Universal Robots PolyScope program: DAS428_958_02_MAR_21_DAS_lado_izquierdo_jig2.urp

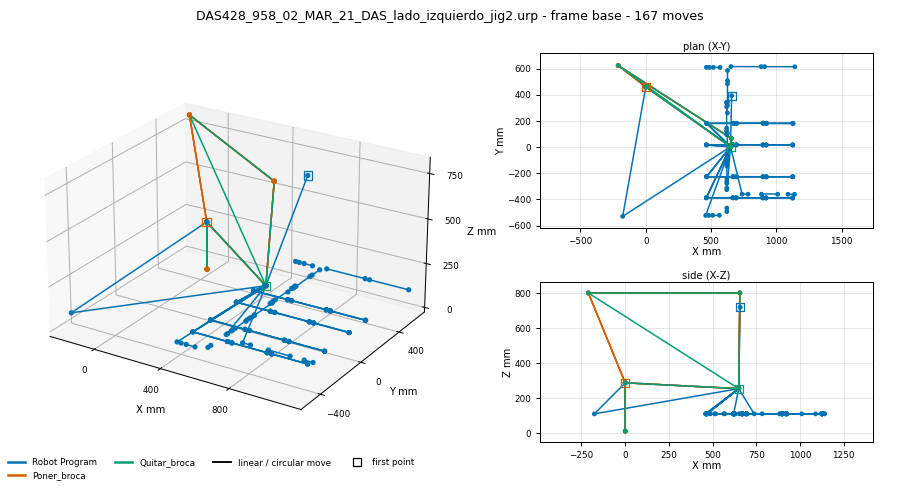
[picture p0: tool path of DAS428_958_02_MAR_21_DAS_lado_izquierdo_jig2.urp in frame base, 167 of 340 moves have a stored position in this frame; points joined in program order, loops and branches not executed]
Program DAS428_958_02_MAR_21_DAS_lado_izquierdo_jig2 (installation=instalacion_derecha_10_MAR_21 directory=/programs/jig2/Izquierda createdIn=5.6.0.90886 lastSavedIn=5.6.0.90886 robotSerialNumber=20195001785)
Calibrated DH parameters: a=[0.000107, -0.568984, -0.552934, -0.00001, -0.000063, 0]; d=[0.180718, -257.998067, 200.685024, 57.48776, 0.119923, 0.115353]; alpha=[1.571119, 0.000876, -0.002498, 1.571178, -1.570523, 0]; deltaTheta=[0, -0.378191, 0.631587, -0.253396, 0, 0]
Robot Program (runOnlyOnce=false)
  Folder Variables
    bajada_broca := p[0,0,-0.008,0,0,0]
    barrenos_menos1 := 0
    barreno_actual := 0
    posicion := p[0,0,300,0,0,0]
    cambiar_broca := False
    barrenos_hechos := 0
    eje7 := 0
    Wait Sleep waitTime=0.5
  Folder Home
    Wait Sleep waitTime=0.3
    MoveL speed 250 mm/s, acceleration 1200 mm/s^2 (useActiveTCP=true) feature=Base
      Waypoint Traslacion: TCP in base x=657.999 y=394.119 z=719.669 mm, rx=0.7459 ry=2.9065 rz=0.0955 rad; joints [-173.083, -83.201, 56.688, 18.113, -333.312, 0.041] deg; TCP offset x=0.411 y=-218.298 z=37.994 mm, rx=1.558 ry=-0.1255 rz=0.1212 rad
      Waypoint Home2: TCP in base x=649.602 y=3.2 z=254.15 mm, rx=-2.4485 ry=-1.9662 rz=-0.0111 rad; joints [-199.372, -96.579, 116.673, -19.801, -286.041, 0.348] deg; TCP offset x=0.411 y=-218.298 z=37.994 mm, rx=1.558 ry=-0.1255 rz=0.1212 rad
      Waypoint Home3: TCP in base x=649.602 y=3.2 z=254.15 mm, rx=-2.4485 ry=-1.9662 rz=-0.0111 rad; joints [-199.372, -96.579, 116.673, -19.801, -286.041, 0.348] deg; TCP offset x=0.411 y=-218.298 z=37.994 mm, rx=1.558 ry=-0.1255 rz=0.1212 rad
      Waypoint Home4: TCP in base x=649.602 y=3.2 z=254.15 mm, rx=-2.4485 ry=-1.9662 rz=-0.0111 rad; joints [-199.372, -96.579, 116.673, -19.801, -286.041, 0.348] deg
      Waypoint PosicionApagado: TCP in base x=-175.961 y=-529.389 z=109.95 mm, rx=0.175 ry=2.1133 rz=-2.1574 rad; joints [-90.111, -89.982, -160.832, -17.508, -269.675, 0.001] deg; TCP offset x=0.411 y=-218.298 z=37.994 mm, rx=1.558 ry=-0.1255 rz=0.1212 rad
      Waypoint Precambio_broca: TCP in base x=0.83 y=461.518 z=287.521 mm, rx=-0.2218 ry=-3.132 rz=0.0004 rad; joints [-125.124, -120.118, 128.54, -7.699, -306.118, -0.232] deg
    SafeHome (positionOptionType=SPEED_AND_ACCELERATION speed=1.047198 acceleration=1.396263 nextMotionTime=2)
    SuppressedNode
      MoveL speed 250 mm/s, acceleration 1200 mm/s^2 (useActiveTCP=true) feature=Base
        Waypoint home_trans: TCP in base x=-171.077 y=546.65 z=109.574 mm, rx=0.1544 ry=3.1247 rz=-0.2011 rad; joints [-91.802, -93.053, 127.954, -27.005, -275.278, -0.192] deg
    Wait Sleep waitTime=0.3
    iniciando_prog := True
    Call Poner_broca
  Folder Posicion2
    Folder Inicio
      eje7 := 2
      MoveL speed 250 mm/s, acceleration 1200 mm/s^2 (useActiveTCP=true) feature=Base
        Waypoint Home2: TCP in base x=649.602 y=3.2 z=254.15 mm, rx=-2.4485 ry=-1.9662 rz=-0.0111 rad; joints [-199.372, -96.579, 116.673, -19.801, -286.041, 0.348] deg; TCP offset x=0.411 y=-218.298 z=37.994 mm, rx=1.558 ry=-0.1255 rz=0.1212 rad
    Folder SeatTracks
      Folder Broca_1
        Folder Linea1
          Folder Marcar_puntos
            MoveL speed 100 mm/s, acceleration 500 mm/s^2 (useActiveTCP=true) feature=Base
              Waypoint Home2: TCP in base x=649.602 y=3.2 z=254.15 mm, rx=-2.4485 ry=-1.9662 rz=-0.0111 rad; joints [-199.372, -96.579, 116.673, -19.801, -286.041, 0.348] deg
              Waypoint Linea1_A: TCP in base x=465.78 y=-226.285 z=110.11 mm, rx=3.1292 ry=0.274 rz=-0.0085 rad; joints [-215.56, -96.678, 133.119, -35.816, -234.732, 0.192] deg; TCP offset x=0.411 y=-218.298 z=37.994 mm, rx=1.558 ry=-0.1255 rz=0.1212 rad
              Waypoint Linea1_B: TCP in base x=669.2 y=-226.066 z=110.222 mm, rx=3.1292 ry=0.2741 rz=-0.0085 rad; joints [-203.814, -77.304, 112.388, -34.338, -222.994, 0.395] deg; TCP offset x=0.411 y=-218.298 z=37.994 mm, rx=1.558 ry=-0.1255 rz=0.1212 rad
              Waypoint Linea1_C: TCP in base x=694.6 y=-226.083 z=110.775 mm, rx=3.1292 ry=0.274 rz=-0.0086 rad; joints [-202.875, -75.175, 109.532, -33.596, -222.053, 0.413] deg
              Waypoint Linea1_D: TCP in base x=897.8 y=-226.331 z=110.549 mm, rx=3.1292 ry=0.2741 rz=-0.0085 rad; joints [-197.398, -58.161, 84.21, -25.204, -216.564, 0.534] deg
              Waypoint Linea1_E: TCP in base x=923.2 y=-226.496 z=110.279 mm, rx=3.1292 ry=0.2741 rz=-0.0086 rad; joints [-196.902, -55.941, 80.587, -23.787, -216.064, 0.545] deg
              Waypoint Linea1_F: TCP in base x=1125.593 y=-226.031 z=110.602 mm, rx=3.1292 ry=0.2741 rz=-0.0087 rad; joints [-193.7, -34.945, 43.134, -7.265, -212.819, 0.625] deg; TCP offset x=0.411 y=-218.298 z=37.994 mm, rx=1.558 ry=-0.1255 rz=0.1212 rad
          Folder AB
            'desbaste_inicial'
            bajada_broca := p[0,0,-0.008,0,0,0]
            barrenos_menos1 := 8
            barreno_actual := 0
            Loop While (checkContinuously=false) expression=barreno_actual≤barrenos_menos1
              Folder Perforacion
                MoveL speed 100 mm/s, acceleration 500 mm/s^2 (useActiveTCP=true) feature=Base
                  internos := interpolate_pose(Linea1_A, Linea1_B, barreno_actual/barrenos_menos1)
                  Waypoint Waypoint (Variable): variable=internos
                  'desbaste_inicial'
                  bajada_broca := p[0,0,-0.008,0,0,0]
                  bajada := p[0,0,0.008,0,0,0]
                  MoveDirectionNode (selectedDirection=ZMinus toolParams=0.015, 0.015)
                    Until DISTANCE (allowActions=false deceleration=3 distanceNodeType=STOP) Distance=0.076; motionParameters(blendRadius=0)
                  Popup Message (haltProgram=false message=punto contacto alanzdo inputType=Text)
                  MoveDirectionNode (selectedDirection=ZPlus toolParams=0.015, 0.015)
                    Until DISTANCE (allowActions=false deceleration=3 distanceNodeType=STOP) Distance=0.002; motionParameters(blendRadius=0)
                  Wait Sleep waitTime=0.3
                  Set DigitalOutput pin=config_out[1]; digitalValue=1
                  Wait Sleep waitTime=0.3
                  Loop Counting (count=3) loopVariable(name=Loop_39)
                    bajar := pose_add(get_actual_tcp_pose(), bajada_broca)
                    Waypoint Waypoint (Variable): motionParameters(jointSpeed=1.047198 jointAcceleration=1.396263 cartesianSpeed=0.001 cartesianAcceleration=0.005); variable=bajar
                    subir := pose_sub(get_actual_tcp_pose(), bajada_broca)
                    Waypoint Waypoint (Variable): motionParameters(jointSpeed=1.047198 jointAcceleration=1.396263 cartesianSpeed=0.005 cartesianAcceleration=0.01); variable=subir
                    bajada_broca := pose_sub(bajada_broca, bajada)
                  MoveDirectionNode (selectedDirection=ZPlus toolParams=0.03, 0.035)
                    Until DISTANCE (allowActions=false deceleration=3 distanceNodeType=STOP) Distance=0.06; motionParameters(blendRadius=0)
                  Set DigitalOutput pin=config_out[1]; digitalValue=0
                  barreno_actual := barreno_actual+1
                  SuppressedNode
                    Call Quitar_broca
                  SuppressedNode
                    Call Poner_broca
          Folder CD
            'desbaste_inicial'
            bajada_broca := p[0,0,-0.008,0,0,0]
            barrenos_menos1 := 8
            barreno_actual := 0
            Loop While (checkContinuously=false) expression=barreno_actual≤barrenos_menos1
              Folder Perforacion
                MoveL speed 100 mm/s, acceleration 500 mm/s^2 (useActiveTCP=true) feature=Base
                  internos := interpolate_pose(Linea1_C, Linea1_D, barreno_actual/barrenos_menos1)
                  Waypoint Waypoint (Variable): variable=internos
                  'desbaste_inicial'
                  bajada_broca := p[0,0,-0.008,0,0,0]
                  bajada := p[0,0,0.008,0,0,0]
                  MoveDirectionNode (selectedDirection=ZMinus toolParams=0.015, 0.015)
                    Until DISTANCE (allowActions=false deceleration=3 distanceNodeType=STOP) Distance=0.076; motionParameters(blendRadius=0)
                  Popup Message (haltProgram=false message=punto contacto alanzdo inputType=Text)
                  MoveDirectionNode (selectedDirection=ZPlus toolParams=0.003, 0.005)
                    Until DISTANCE (allowActions=false deceleration=3 distanceNodeType=STOP) Distance=0.002; motionParameters(blendRadius=0)
                  Wait Sleep waitTime=0.3
                  Set DigitalOutput pin=config_out[1]; digitalValue=1
                  Wait Sleep waitTime=0.3
                  Loop Counting (count=3) loopVariable(name=Loop_56)
                    bajar := pose_add(get_actual_tcp_pose(), bajada_broca)
                    Waypoint Waypoint (Variable): motionParameters(jointSpeed=1.047198 jointAcceleration=1.396263 cartesianSpeed=0.001 cartesianAcceleration=0.005); variable=bajar
                    subir := pose_sub(get_actual_tcp_pose(), bajada_broca)
                    Waypoint Waypoint (Variable): motionParameters(jointSpeed=1.047198 jointAcceleration=1.396263 cartesianSpeed=0.005 cartesianAcceleration=0.01); variable=subir
                    bajada_broca := pose_sub(bajada_broca, bajada)
                  MoveDirectionNode (selectedDirection=ZPlus toolParams=0.03, 0.035)
                    Until DISTANCE (allowActions=false deceleration=3 distanceNodeType=STOP) Distance=0.06; motionParameters(blendRadius=0)
                  Set DigitalOutput pin=config_out[1]; digitalValue=0
                  barreno_actual := barreno_actual+1
                  SuppressedNode
                    Call Quitar_broca
                  SuppressedNode
                    Call Poner_broca
          Folder EF
            'desbaste_inicial'
            bajada_broca := p[0,0,-0.008,0,0,0]
            barrenos_menos1 := 8
            barreno_actual := 0
            Loop While (checkContinuously=false) expression=barreno_actual≤barrenos_menos1
              Folder Perforacion
                MoveL speed 100 mm/s, acceleration 500 mm/s^2 (useActiveTCP=true) feature=Base
                  internos := interpolate_pose(Linea1_E, Linea1_F, barreno_actual/barrenos_menos1)
                  Waypoint Waypoint (Variable): variable=internos
                  'desbaste_inicial'
                  bajada_broca := p[0,0,-0.008,0,0,0]
                  bajada := p[0,0,0.008,0,0,0]
                  MoveDirectionNode (selectedDirection=ZMinus toolParams=0.015, 0.015)
                    Until DISTANCE (allowActions=false deceleration=3 distanceNodeType=STOP) Distance=0.076; motionParameters(blendRadius=0)
                  Popup Message (haltProgram=false message=punto contacto alanzdo inputType=Text)
                  MoveDirectionNode (selectedDirection=ZPlus toolParams=0.003, 0.005)
                    Until DISTANCE (allowActions=false deceleration=3 distanceNodeType=STOP) Distance=0.002; motionParameters(blendRadius=0)
                  Wait Sleep waitTime=0.3
                  Set DigitalOutput pin=config_out[1]; digitalValue=1
                  Wait Sleep waitTime=0.3
                  Loop Counting (count=3) loopVariable(name=Loop_61)
                    bajar := pose_add(get_actual_tcp_pose(), bajada_broca)
                    Waypoint Waypoint (Variable): motionParameters(jointSpeed=1.047198 jointAcceleration=1.396263 cartesianSpeed=0.001 cartesianAcceleration=0.005); variable=bajar
                    subir := pose_sub(get_actual_tcp_pose(), bajada_broca)
                    Waypoint Waypoint (Variable): motionParameters(jointSpeed=1.047198 jointAcceleration=1.396263 cartesianSpeed=0.005 cartesianAcceleration=0.01); variable=subir
                    bajada_broca := pose_sub(bajada_broca, bajada)
                  MoveDirectionNode (selectedDirection=ZPlus toolParams=0.03, 0.035)
                    Until DISTANCE (allowActions=false deceleration=3 distanceNodeType=STOP) Distance=0.06; motionParameters(blendRadius=0)
                  Set DigitalOutput pin=config_out[1]; digitalValue=0
                  barreno_actual := barreno_actual+1
                  SuppressedNode
                    Call Quitar_broca
                  SuppressedNode
                    Call Poner_broca
        Popup Message (haltProgram=false message=Linea1 con chica Terminada! inputType=Text)
        Folder Linea2
          Folder Marcar_puntos
            MoveL speed 100 mm/s, acceleration 500 mm/s^2 (useActiveTCP=true) feature=Base
              Waypoint Home2: TCP in base x=649.602 y=3.2 z=254.15 mm, rx=-2.4485 ry=-1.9662 rz=-0.0111 rad; joints [-199.372, -96.579, 116.673, -19.801, -286.041, 0.348] deg; TCP offset x=0.411 y=-218.298 z=37.994 mm, rx=1.558 ry=-0.1255 rz=0.1212 rad
              Waypoint Linea2_A: TCP in base x=466.954 y=182.157 z=110.172 mm, rx=-2.4485 ry=-1.9662 rz=-0.0111 rad; joints [-177.403, -103.734, 138.62, -34.639, -264.097, 0.47] deg; TCP offset x=0.411 y=-218.298 z=37.994 mm, rx=1.558 ry=-0.1255 rz=0.1212 rad
              Waypoint Linea2_B: TCP in base x=671.81 y=182.878 z=110.175 mm, rx=-2.4484 ry=-1.9662 rz=-0.011 rad; joints [-178.316, -83.76, 120.353, -36.338, -265.022, 0.484] deg; TCP offset x=0.411 y=-218.298 z=37.994 mm, rx=1.558 ry=-0.1255 rz=0.1212 rad
              Waypoint Linea2_C: TCP in base x=694.981 y=182.77 z=110.46 mm, rx=-2.4483 ry=-1.9662 rz=-0.0109 rad; joints [-178.397, -81.801, 118.029, -35.97, -265.106, 0.486] deg; TCP offset x=0.411 y=-218.298 z=37.994 mm, rx=1.558 ry=-0.1255 rz=0.1212 rad
              Waypoint Linea2_D: TCP in base x=898.787 y=183.235 z=110.403 mm, rx=-2.4483 ry=-1.9664 rz=-0.011 rad; joints [-178.787, -65.181, 95.382, -29.948, -265.491, 0.487] deg
              Waypoint Linea2_E: TCP in base x=923.79 y=182.507 z=110.324 mm, rx=-2.4483 ry=-1.9664 rz=-0.011 rad; joints [-178.879, -63.164, 92.292, -28.877, -265.58, 0.486] deg
              Waypoint Linea2_F: TCP in base x=1126.946 y=182.371 z=110.084 mm, rx=-2.4483 ry=-1.9664 rz=-0.011 rad; joints [-179.118, -45.199, 62.135, -16.683, -265.793, 0.483] deg
          Folder AB
            'desbaste_inicial'
            bajada_broca := p[0,0,-0.008,0,0,0]
            barrenos_menos1 := 8
            barreno_actual := 0
            Loop While (checkContinuously=false) expression=barreno_actual≤barrenos_menos1
              Folder Perforacion
                MoveL speed 100 mm/s, acceleration 500 mm/s^2 (useActiveTCP=true) feature=Base
                  internos := interpolate_pose(Linea2_A, Linea2_B, barreno_actual/barrenos_menos1)
                  Waypoint Waypoint (Variable): variable=internos
                  'desbaste_inicial'
                  bajada_broca := p[0,0,-0.008,0,0,0]
                  bajada := p[0,0,0.008,0,0,0]
                  MoveDirectionNode (selectedDirection=ZMinus toolParams=0.015, 0.015)
                    Until DISTANCE (allowActions=false deceleration=3 distanceNodeType=STOP) Distance=0.076; motionParameters(blendRadius=0)
                  Popup Message (haltProgram=false message=punto contacto alanzdo inputType=Text)
                  MoveDirectionNode (selectedDirection=ZPlus toolParams=0.003, 0.005)
                    Until DISTANCE (allowActions=false deceleration=3 distanceNodeType=STOP) Distance=0.002; motionParameters(blendRadius=0)
                  Wait Sleep waitTime=0.3
                  Set DigitalOutput pin=config_out[1]; digitalValue=1
                  Wait Sleep waitTime=0.3
                  Loop Counting (count=3) loopVariable(name=Loop_63)
                    bajar := pose_add(get_actual_tcp_pose(), bajada_broca)
                    Waypoint Waypoint (Variable): motionParameters(jointSpeed=1.047198 jointAcceleration=1.396263 cartesianSpeed=0.001 cartesianAcceleration=0.005); variable=bajar
                    subir := pose_sub(get_actual_tcp_pose(), bajada_broca)
                    Waypoint Waypoint (Variable): motionParameters(jointSpeed=1.047198 jointAcceleration=1.396263 cartesianSpeed=0.005 cartesianAcceleration=0.01); variable=subir
                    bajada_broca := pose_sub(bajada_broca, bajada)
                  MoveDirectionNode (selectedDirection=ZPlus toolParams=0.03, 0.035)
                    Until DISTANCE (allowActions=false deceleration=3 distanceNodeType=STOP) Distance=0.06; motionParameters(blendRadius=0)
                  Set DigitalOutput pin=config_out[1]; digitalValue=0
                  barreno_actual := barreno_actual+1
                  SuppressedNode
                    Call Quitar_broca
                  SuppressedNode
                    Call Poner_broca
          Folder CD
            'desbaste_inicial'
            bajada_broca := p[0,0,-0.008,0,0,0]
            barrenos_menos1 := 8
            barreno_actual := 0
            Loop While (checkContinuously=false) expression=barreno_actual≤barrenos_menos1
              Folder Perforacion
                MoveL speed 100 mm/s, acceleration 500 mm/s^2 (useActiveTCP=true) feature=Base
                  internos := interpolate_pose(Linea2_C, Linea2_D, barreno_actual/barrenos_menos1)
                  Waypoint Waypoint (Variable): variable=internos
                  'desbaste_inicial'
                  bajada_broca := p[0,0,-0.008,0,0,0]
                  bajada := p[0,0,0.008,0,0,0]
                  MoveDirectionNode (selectedDirection=ZMinus toolParams=0.015, 0.015)
                    Until DISTANCE (allowActions=false deceleration=3 distanceNodeType=STOP) Distance=0.076; motionParameters(blendRadius=0)
                  Popup Message (haltProgram=false message=punto contacto alanzdo inputType=Text)
                  MoveDirectionNode (selectedDirection=ZPlus toolParams=0.003, 0.005)
                    Until DISTANCE (allowActions=false deceleration=3 distanceNodeType=STOP) Distance=0.002; motionParameters(blendRadius=0)
                  Wait Sleep waitTime=0.3
                  Set DigitalOutput pin=config_out[1]; digitalValue=1
                  Wait Sleep waitTime=0.3
                  Loop Counting (count=3) loopVariable(name=Loop_65)
                    bajar := pose_add(get_actual_tcp_pose(), bajada_broca)
                    Waypoint Waypoint (Variable): motionParameters(jointSpeed=1.047198 jointAcceleration=1.396263 cartesianSpeed=0.001 cartesianAcceleration=0.005); variable=bajar
                    subir := pose_sub(get_actual_tcp_pose(), bajada_broca)
                    Waypoint Waypoint (Variable): motionParameters(jointSpeed=1.047198 jointAcceleration=1.396263 cartesianSpeed=0.005 cartesianAcceleration=0.01); variable=subir
                    bajada_broca := pose_sub(bajada_broca, bajada)
                  MoveDirectionNode (selectedDirection=ZPlus toolParams=0.03, 0.035)
                    Until DISTANCE (allowActions=false deceleration=3 distanceNodeType=STOP) Distance=0.06; motionParameters(blendRadius=0)
                  Set DigitalOutput pin=config_out[1]; digitalValue=0
                  barreno_actual := barreno_actual+1
                  SuppressedNode
                    Call Quitar_broca
                  SuppressedNode
                    Call Poner_broca
          Folder EF
            'desbaste_inicial'
            bajada_broca := p[0,0,-0.008,0,0,0]
            barrenos_menos1 := 8
            barreno_actual := 0
            Loop While (checkContinuously=false) expression=barreno_actual≤barrenos_menos1
              Folder Perforacion
                MoveL speed 100 mm/s, acceleration 500 mm/s^2 (useActiveTCP=true) feature=Base
                  internos := interpolate_pose(Linea2_E, Linea2_F, barreno_actual/barrenos_menos1)
                  Waypoint Waypoint (Variable): variable=internos
                  'desbaste_inicial'
                  bajada_broca := p[0,0,-0.008,0,0,0]
                  bajada := p[0,0,0.008,0,0,0]
                  MoveDirectionNode (selectedDirection=ZMinus toolParams=0.015, 0.015)
                    Until DISTANCE (allowActions=false deceleration=3 distanceNodeType=STOP) Distance=0.076; motionParameters(blendRadius=0)
                  Popup Message (haltProgram=false message=punto contacto alanzdo inputType=Text)
                  MoveDirectionNode (selectedDirection=ZPlus toolParams=0.003, 0.005)
                    Until DISTANCE (allowActions=false deceleration=3 distanceNodeType=STOP) Distance=0.002; motionParameters(blendRadius=0)
                  Wait Sleep waitTime=0.3
                  Set DigitalOutput pin=config_out[1]; digitalValue=1
                  Wait Sleep waitTime=0.3
                  Loop Counting (count=3) loopVariable(name=Loop_67)
                    bajar := pose_add(get_actual_tcp_pose(), bajada_broca)
                    Waypoint Waypoint (Variable): motionParameters(jointSpeed=1.047198 jointAcceleration=1.396263 cartesianSpeed=0.001 cartesianAcceleration=0.005); variable=bajar
                    subir := pose_sub(get_actual_tcp_pose(), bajada_broca)
                    Waypoint Waypoint (Variable): motionParameters(jointSpeed=1.047198 jointAcceleration=1.396263 cartesianSpeed=0.005 cartesianAcceleration=0.01); variable=subir
                    bajada_broca := pose_sub(bajada_broca, bajada)
                  MoveDirectionNode (selectedDirection=ZPlus toolParams=0.03, 0.035)
                    Until DISTANCE (allowActions=false deceleration=3 distanceNodeType=STOP) Distance=0.06; motionParameters(blendRadius=0)
                  Set DigitalOutput pin=config_out[1]; digitalValue=0
                  barreno_actual := barreno_actual+1
                  If barreno_actual≥barrenos_menos1
                    cambiar_broca := True
                  SuppressedNode
                    Call Quitar_broca
                  SuppressedNode
                    Call Poner_broca
        Popup Message (haltProgram=false message=Linea2 con chica Terminada! inputType=Text)
      Folder Broca_2
        Folder Linea1
          Folder Marcar_puntos
            MoveL speed 100 mm/s, acceleration 500 mm/s^2 (useActiveTCP=true) feature=Base
              Waypoint Home2: TCP in base x=649.602 y=3.2 z=254.15 mm, rx=-2.4485 ry=-1.9662 rz=-0.0111 rad; joints [-199.372, -96.579, 116.673, -19.801, -286.041, 0.348] deg; TCP offset x=0.411 y=-218.298 z=37.994 mm, rx=1.558 ry=-0.1255 rz=0.1212 rad
              Waypoint Linea1_A: TCP in base x=465.78 y=-226.285 z=110.11 mm, rx=3.1292 ry=0.274 rz=-0.0085 rad; joints [-215.56, -96.678, 133.119, -35.816, -234.732, 0.192] deg; TCP offset x=0.411 y=-218.298 z=37.994 mm, rx=1.558 ry=-0.1255 rz=0.1212 rad
              Waypoint Linea1_B: TCP in base x=669.2 y=-226.066 z=110.222 mm, rx=3.1292 ry=0.2741 rz=-0.0085 rad; joints [-203.814, -77.304, 112.388, -34.338, -222.994, 0.395] deg; TCP offset x=0.411 y=-218.298 z=37.994 mm, rx=1.558 ry=-0.1255 rz=0.1212 rad
              Waypoint Linea1_C: TCP in base x=694.6 y=-226.083 z=110.775 mm, rx=3.1292 ry=0.274 rz=-0.0086 rad; joints [-202.875, -75.175, 109.532, -33.596, -222.053, 0.413] deg
              Waypoint Linea1_D: TCP in base x=897.8 y=-226.331 z=110.549 mm, rx=3.1292 ry=0.2741 rz=-0.0085 rad; joints [-197.398, -58.161, 84.21, -25.204, -216.564, 0.534] deg
              Waypoint Linea1_E: TCP in base x=923.2 y=-226.496 z=110.279 mm, rx=3.1292 ry=0.2741 rz=-0.0086 rad; joints [-196.902, -55.941, 80.587, -23.787, -216.064, 0.545] deg
              Waypoint Linea1_F: TCP in base x=1125.593 y=-226.031 z=110.602 mm, rx=3.1292 ry=0.2741 rz=-0.0087 rad; joints [-193.7, -34.945, 43.134, -7.265, -212.819, 0.625] deg; TCP offset x=0.411 y=-218.298 z=37.994 mm, rx=1.558 ry=-0.1255 rz=0.1212 rad
          Folder AB
            'desbaste_inicial'
            bajada_broca := p[0,0,-0.012,0,0,0]
            barrenos_menos1 := 8
            barreno_actual := 0
            Loop While (checkContinuously=false) expression=barreno_actual≤barrenos_menos1
              Folder Perforacion
                MoveL speed 100 mm/s, acceleration 500 mm/s^2 (useActiveTCP=true) feature=Base
                  internos := interpolate_pose(Linea1_A, Linea1_B, barreno_actual/barrenos_menos1)
                  Waypoint Waypoint (Variable): variable=internos
                  'desbaste_inicial'
                  bajada_broca := p[0,0,-0.012,0,0,0]
                  bajada := p[0,0,0.012,0,0,0]
                  MoveDirectionNode (selectedDirection=ZMinus toolParams=0.015, 0.015)
                    Until DISTANCE (allowActions=false deceleration=3 distanceNodeType=STOP) Distance=0.076; motionParameters(blendRadius=0)
                  Popup Message (haltProgram=false message=punto contacto alanzdo inputType=Text)
                  MoveDirectionNode (selectedDirection=ZPlus toolParams=0.003, 0.005)
                    Until DISTANCE (allowActions=false deceleration=3 distanceNodeType=STOP) Distance=0.002; motionParameters(blendRadius=0)
                  Wait Sleep waitTime=0.3
                  Set DigitalOutput pin=config_out[1]; digitalValue=1
                  Wait Sleep waitTime=0.3
                  Loop Counting (count=2) loopVariable(name=Loop_69)
                    bajar := pose_add(get_actual_tcp_pose(), bajada_broca)
                    Waypoint Waypoint (Variable): motionParameters(jointSpeed=1.047198 jointAcceleration=1.396263 cartesianSpeed=0.001 cartesianAcceleration=0.005); variable=bajar
                    subir := pose_sub(get_actual_tcp_pose(), bajada_broca)
                    Waypoint Waypoint (Variable): motionParameters(jointSpeed=1.047198 jointAcceleration=1.396263 cartesianSpeed=0.005 cartesianAcceleration=0.01); variable=subir
                    bajada_broca := pose_sub(bajada_broca, bajada)
                  MoveDirectionNode (selectedDirection=ZPlus toolParams=0.03, 0.035)
                    Until DISTANCE (allowActions=false deceleration=3 distanceNodeType=STOP) Distance=0.06; motionParameters(blendRadius=0)
                  Set DigitalOutput pin=config_out[1]; digitalValue=0
                  barreno_actual := barreno_actual+1
                  Call Quitar_broca
                  Call Poner_broca
          Folder CD
            'desbaste_inicial'
            bajada_broca := p[0,0,-0.012,0,0,0]
            barrenos_menos1 := 8
            barreno_actual := 0
            Loop While (checkContinuously=false) expression=barreno_actual≤barrenos_menos1
              Folder Perforacion
                MoveL speed 100 mm/s, acceleration 500 mm/s^2 (useActiveTCP=true) feature=Base
                  internos := interpolate_pose(Linea1_C, Linea1_D, barreno_actual/barrenos_menos1)
                  Waypoint Waypoint (Variable): variable=internos
                  'desbaste_inicial'
                  bajada_broca := p[0,0,-0.012,0,0,0]
                  bajada := p[0,0,0.012,0,0,0]
                  MoveDirectionNode (selectedDirection=ZMinus toolParams=0.015, 0.015)
                    Until DISTANCE (allowActions=false deceleration=3 distanceNodeType=STOP) Distance=0.076; motionParameters(blendRadius=0)
                  Popup Message (haltProgram=false message=punto contacto alanzdo inputType=Text)
                  MoveDirectionNode (selectedDirection=ZPlus toolParams=0.003, 0.005)
                    Until DISTANCE (allowActions=false deceleration=3 distanceNodeType=STOP) Distance=0.002; motionParameters(blendRadius=0)
                  Wait Sleep waitTime=0.3
                  Set DigitalOutput pin=config_out[1]; digitalValue=1
                  Wait Sleep waitTime=0.3
                  Loop Counting (count=2) loopVariable(name=Loop_71)
                    bajar := pose_add(get_actual_tcp_pose(), bajada_broca)
                    Waypoint Waypoint (Variable): motionParameters(jointSpeed=1.047198 jointAcceleration=1.396263 cartesianSpeed=0.001 cartesianAcceleration=0.005); variable=bajar
                    subir := pose_sub(get_actual_tcp_pose(), bajada_broca)
                    Waypoint Waypoint (Variable): motionParameters(jointSpeed=1.047198 jointAcceleration=1.396263 cartesianSpeed=0.005 cartesianAcceleration=0.01); variable=subir
                    bajada_broca := pose_sub(bajada_broca, bajada)
                  MoveDirectionNode (selectedDirection=ZPlus toolParams=0.03, 0.035)
                    Until DISTANCE (allowActions=false deceleration=3 distanceNodeType=STOP) Distance=0.06; motionParameters(blendRadius=0)
                  Set DigitalOutput pin=config_out[1]; digitalValue=0
                  barreno_actual := barreno_actual+1
                  Call Quitar_broca
                  Call Poner_broca
          Folder EF
            'desbaste_inicial'
            bajada_broca := p[0,0,-0.012,0,0,0]
            barrenos_menos1 := 8
            barreno_actual := 0
            Loop While (checkContinuously=false) expression=barreno_actual≤barrenos_menos1
              Folder Perforacion
                MoveL speed 100 mm/s, acceleration 500 mm/s^2 (useActiveTCP=true) feature=Base
                  internos := interpolate_pose(Linea1_E, Linea1_F, barreno_actual/barrenos_menos1)
                  Waypoint Waypoint (Variable): variable=internos
                  'desbaste_inicial'
                  bajada_broca := p[0,0,-0.012,0,0,0]
                  bajada := p[0,0,0.012,0,0,0]
                  MoveDirectionNode (selectedDirection=ZMinus toolParams=0.015, 0.015)
                    Until DISTANCE (allowActions=false deceleration=3 distanceNodeType=STOP) Distance=0.076; motionParameters(blendRadius=0)
                  Popup Message (haltProgram=false message=punto contacto alanzdo inputType=Text)
                  MoveDirectionNode (selectedDirection=ZPlus toolParams=0.003, 0.005)
                    Until DISTANCE (allowActions=false deceleration=3 distanceNodeType=STOP) Distance=0.002; motionParameters(blendRadius=0)
                  Wait Sleep waitTime=0.3
                  Set DigitalOutput pin=config_out[1]; digitalValue=1
                  Wait Sleep waitTime=0.3
                  Loop Counting (count=2) loopVariable(name=Loop_73)
                    bajar := pose_add(get_actual_tcp_pose(), bajada_broca)
                    Waypoint Waypoint (Variable): motionParameters(jointSpeed=1.047198 jointAcceleration=1.396263 cartesianSpeed=0.001 cartesianAcceleration=0.005); variable=bajar
                    subir := pose_sub(get_actual_tcp_pose(), bajada_broca)
                    Waypoint Waypoint (Variable): motionParameters(jointSpeed=1.047198 jointAcceleration=1.396263 cartesianSpeed=0.005 cartesianAcceleration=0.01); variable=subir
                    bajada_broca := pose_sub(bajada_broca, bajada)
                  MoveDirectionNode (selectedDirection=ZPlus toolParams=0.03, 0.035)
                    Until DISTANCE (allowActions=false deceleration=3 distanceNodeType=STOP) Distance=0.06; motionParameters(blendRadius=0)
                  Set DigitalOutput pin=config_out[1]; digitalValue=0
                  barreno_actual := barreno_actual+1
                  Call Quitar_broca
                  Call Poner_broca
        Popup Message (haltProgram=false message=Linea1 con media Terminada! inputType=Text)
        Folder Linea2
          Folder Marcar_puntos
            MoveL speed 100 mm/s, acceleration 500 mm/s^2 (useActiveTCP=true) feature=Base
              Waypoint Home2: TCP in base x=649.602 y=3.2 z=254.15 mm, rx=-2.4485 ry=-1.9662 rz=-0.0111 rad; joints [-199.372, -96.579, 116.673, -19.801, -286.041, 0.348] deg; TCP offset x=0.411 y=-218.298 z=37.994 mm, rx=1.558 ry=-0.1255 rz=0.1212 rad
              Waypoint Linea2_A: TCP in base x=466.954 y=182.157 z=110.172 mm, rx=-2.4485 ry=-1.9662 rz=-0.0111 rad; joints [-177.403, -103.734, 138.62, -34.639, -264.097, 0.47] deg; TCP offset x=0.411 y=-218.298 z=37.994 mm, rx=1.558 ry=-0.1255 rz=0.1212 rad
              Waypoint Linea2_B: TCP in base x=671.81 y=182.878 z=110.175 mm, rx=-2.4484 ry=-1.9662 rz=-0.011 rad; joints [-178.316, -83.76, 120.353, -36.338, -265.022, 0.484] deg; TCP offset x=0.411 y=-218.298 z=37.994 mm, rx=1.558 ry=-0.1255 rz=0.1212 rad
              Waypoint Linea2_C: TCP in base x=694.981 y=182.77 z=110.46 mm, rx=-2.4483 ry=-1.9662 rz=-0.0109 rad; joints [-178.397, -81.801, 118.029, -35.97, -265.106, 0.486] deg; TCP offset x=0.411 y=-218.298 z=37.994 mm, rx=1.558 ry=-0.1255 rz=0.1212 rad
              Waypoint Linea2_D: TCP in base x=898.787 y=183.235 z=110.403 mm, rx=-2.4483 ry=-1.9664 rz=-0.011 rad; joints [-178.787, -65.181, 95.382, -29.948, -265.491, 0.487] deg
              Waypoint Linea2_E: TCP in base x=923.79 y=182.507 z=110.324 mm, rx=-2.4483 ry=-1.9664 rz=-0.011 rad; joints [-178.879, -63.164, 92.292, -28.877, -265.58, 0.486] deg
              Waypoint Linea2_F: TCP in base x=1126.946 y=182.371 z=110.084 mm, rx=-2.4483 ry=-1.9664 rz=-0.011 rad; joints [-179.118, -45.199, 62.135, -16.683, -265.793, 0.483] deg
          Folder AB
            'desbaste_inicial'
            bajada_broca := p[0,0,-0.012,0,0,0]
            barrenos_menos1 := 8
            barreno_actual := 0
            Loop While (checkContinuously=false) expression=barreno_actual≤barrenos_menos1
              Folder Perforacion
                MoveL speed 100 mm/s, acceleration 500 mm/s^2 (useActiveTCP=true) feature=Base
                  internos := interpolate_pose(Linea2_A, Linea2_B, barreno_actual/barrenos_menos1)
                  Waypoint Waypoint (Variable): variable=internos
                  'desbaste_inicial'
                  bajada_broca := p[0,0,-0.012,0,0,0]
                  bajada := p[0,0,0.012,0,0,0]
                  MoveDirectionNode (selectedDirection=ZMinus toolParams=0.015, 0.015)
                    Until DISTANCE (allowActions=false deceleration=3 distanceNodeType=STOP) Distance=0.076; motionParameters(blendRadius=0)
                  Popup Message (haltProgram=false message=punto contacto alanzdo inputType=Text)
                  MoveDirectionNode (selectedDirection=ZPlus toolParams=0.003, 0.005)
                    Until DISTANCE (allowActions=false deceleration=3 distanceNodeType=STOP) Distance=0.002; motionParameters(blendRadius=0)
                  Wait Sleep waitTime=0.3
                  Set DigitalOutput pin=config_out[1]; digitalValue=1
                  Wait Sleep waitTime=0.3
                  Loop Counting (count=2) loopVariable(name=Loop_75)
                    bajar := pose_add(get_actual_tcp_pose(), bajada_broca)
                    Waypoint Waypoint (Variable): motionParameters(jointSpeed=1.047198 jointAcceleration=1.396263 cartesianSpeed=0.001 cartesianAcceleration=0.005); variable=bajar
                    subir := pose_sub(get_actual_tcp_pose(), bajada_broca)
                    Waypoint Waypoint (Variable): motionParameters(jointSpeed=1.047198 jointAcceleration=1.396263 cartesianSpeed=0.005 cartesianAcceleration=0.01); variable=subir
                    bajada_broca := pose_sub(bajada_broca, bajada)
                  MoveDirectionNode (selectedDirection=ZPlus toolParams=0.03, 0.035)
                    Until DISTANCE (allowActions=false deceleration=3 distanceNodeType=STOP) Distance=0.06; motionParameters(blendRadius=0)
                  Set DigitalOutput pin=config_out[1]; digitalValue=0
                  barreno_actual := barreno_actual+1
                  Call Quitar_broca
                  Call Poner_broca
          Folder CD
            'desbaste_inicial'
            bajada_broca := p[0,0,-0.012,0,0,0]
            barrenos_menos1 := 8
            barreno_actual := 0
            Loop While (checkContinuously=false) expression=barreno_actual≤barrenos_menos1
              Folder Perforacion
                MoveL speed 100 mm/s, acceleration 500 mm/s^2 (useActiveTCP=true) feature=Base
                  internos := interpolate_pose(Linea2_C, Linea2_D, barreno_actual/barrenos_menos1)
                  Waypoint Waypoint (Variable): variable=internos
                  'desbaste_inicial'
                  bajada_broca := p[0,0,-0.012,0,0,0]
                  bajada := p[0,0,0.012,0,0,0]
                  MoveDirectionNode (selectedDirection=ZMinus toolParams=0.015, 0.015)
                    Until DISTANCE (allowActions=false deceleration=3 distanceNodeType=STOP) Distance=0.076; motionParameters(blendRadius=0)
                  Popup Message (haltProgram=false message=punto contacto alanzdo inputType=Text)
                  MoveDirectionNode (selectedDirection=ZPlus toolParams=0.003, 0.005)
                    Until DISTANCE (allowActions=false deceleration=3 distanceNodeType=STOP) Distance=0.002; motionParameters(blendRadius=0)
                  Wait Sleep waitTime=0.3
                  Set DigitalOutput pin=config_out[1]; digitalValue=1
                  Wait Sleep waitTime=0.3
                  Loop Counting (count=2) loopVariable(name=Loop_78)
                    bajar := pose_add(get_actual_tcp_pose(), bajada_broca)
                    Waypoint Waypoint (Variable): motionParameters(jointSpeed=1.047198 jointAcceleration=1.396263 cartesianSpeed=0.001 cartesianAcceleration=0.005); variable=bajar
                    subir := pose_sub(get_actual_tcp_pose(), bajada_broca)
                    Waypoint Waypoint (Variable): motionParameters(jointSpeed=1.047198 jointAcceleration=1.396263 cartesianSpeed=0.005 cartesianAcceleration=0.01); variable=subir
                    bajada_broca := pose_sub(bajada_broca, bajada)
                  MoveDirectionNode (selectedDirection=ZPlus toolParams=0.03, 0.035)
                    Until DISTANCE (allowActions=false deceleration=3 distanceNodeType=STOP) Distance=0.06; motionParameters(blendRadius=0)
                  Set DigitalOutput pin=config_out[1]; digitalValue=0
                  barreno_actual := barreno_actual+1
                  Call Quitar_broca
                  Call Poner_broca
          Folder EF
            'desbaste_inicial'
            bajada_broca := p[0,0,-0.012,0,0,0]
            barrenos_menos1 := 8
            barreno_actual := 0
            Loop While (checkContinuously=false) expression=barreno_actual≤barrenos_menos1
              Folder Perforacion
                MoveL speed 100 mm/s, acceleration 500 mm/s^2 (useActiveTCP=true) feature=Base
                  internos := interpolate_pose(Linea2_E, Linea2_F, barreno_actual/barrenos_menos1)
                  Waypoint Waypoint (Variable): variable=internos
                  'desbaste_inicial'
                  bajada_broca := p[0,0,-0.012,0,0,0]
                  bajada := p[0,0,0.012,0,0,0]
                  MoveDirectionNode (selectedDirection=ZMinus toolParams=0.015, 0.015)
                    Until DISTANCE (allowActions=false deceleration=3 distanceNodeType=STOP) Distance=0.076; motionParameters(blendRadius=0)
                  Popup Message (haltProgram=false message=punto contacto alanzdo inputType=Text)
                  MoveDirectionNode (selectedDirection=ZPlus toolParams=0.003, 0.005)
                    Until DISTANCE (allowActions=false deceleration=3 distanceNodeType=STOP) Distance=0.002; motionParameters(blendRadius=0)
                  Wait Sleep waitTime=0.3
                  Set DigitalOutput pin=config_out[1]; digitalValue=1
                  Wait Sleep waitTime=0.3
                  Loop Counting (count=2) loopVariable(name=Loop_80)
                    bajar := pose_add(get_actual_tcp_pose(), bajada_broca)
                    Waypoint Waypoint (Variable): motionParameters(jointSpeed=1.047198 jointAcceleration=1.396263 cartesianSpeed=0.001 cartesianAcceleration=0.005); variable=bajar
                    subir := pose_sub(get_actual_tcp_pose(), bajada_broca)
                    Waypoint Waypoint (Variable): motionParameters(jointSpeed=1.047198 jointAcceleration=1.396263 cartesianSpeed=0.005 cartesianAcceleration=0.01); variable=subir
                    bajada_broca := pose_sub(bajada_broca, bajada)
                  MoveDirectionNode (selectedDirection=ZPlus toolParams=0.03, 0.035)
                    Until DISTANCE (allowActions=false deceleration=3 distanceNodeType=STOP) Distance=0.06; motionParameters(blendRadius=0)
                  Set DigitalOutput pin=config_out[1]; digitalValue=0
                  barreno_actual := barreno_actual+1
                  If barreno_actual≥barrenos_menos1
                    cambiar_broca := True
                  Call Quitar_broca
                  Call Poner_broca
        Popup Message (haltProgram=false message=Linea2 con media Terminada! inputType=Text)
      Folder Broca_3
        Folder Linea1
          Folder Marcar_puntos
            MoveL speed 100 mm/s, acceleration 500 mm/s^2 (useActiveTCP=true) feature=Base
              Waypoint Home2: TCP in base x=649.602 y=3.2 z=254.15 mm, rx=-2.4485 ry=-1.9662 rz=-0.0111 rad; joints [-199.372, -96.579, 116.673, -19.801, -286.041, 0.348] deg; TCP offset x=0.411 y=-218.298 z=37.994 mm, rx=1.558 ry=-0.1255 rz=0.1212 rad
              Folder var
                barrenos_hechos := 2
                eje7 := 2
                cambiar_broca := False
                iniciando_prog := False
              Waypoint Linea1_A: TCP in base x=465.78 y=-226.285 z=110.11 mm, rx=3.1292 ry=0.274 rz=-0.0085 rad; joints [-215.56, -96.678, 133.119, -35.816, -234.732, 0.192] deg; TCP offset x=0.411 y=-218.298 z=37.994 mm, rx=1.558 ry=-0.1255 rz=0.1212 rad
              Waypoint Linea1_B: TCP in base x=669.2 y=-226.066 z=110.222 mm, rx=3.1292 ry=0.2741 rz=-0.0085 rad; joints [-203.814, -77.304, 112.388, -34.338, -222.994, 0.395] deg; TCP offset x=0.411 y=-218.298 z=37.994 mm, rx=1.558 ry=-0.1255 rz=0.1212 rad
              Waypoint Linea1_C: TCP in base x=694.6 y=-226.083 z=110.775 mm, rx=3.1292 ry=0.274 rz=-0.0086 rad; joints [-202.875, -75.175, 109.532, -33.596, -222.053, 0.413] deg
              Waypoint Linea1_D: TCP in base x=897.8 y=-226.331 z=110.549 mm, rx=3.1292 ry=0.2741 rz=-0.0085 rad; joints [-197.398, -58.161, 84.21, -25.204, -216.564, 0.534] deg
              Waypoint Linea1_E: TCP in base x=923.2 y=-226.496 z=110.279 mm, rx=3.1292 ry=0.2741 rz=-0.0086 rad; joints [-196.902, -55.941, 80.587, -23.787, -216.064, 0.545] deg
              Waypoint Linea1_F: TCP in base x=1125.593 y=-226.031 z=110.602 mm, rx=3.1292 ry=0.2741 rz=-0.0087 rad; joints [-193.7, -34.945, 43.134, -7.265, -212.819, 0.625] deg; TCP offset x=0.411 y=-218.298 z=37.994 mm, rx=1.558 ry=-0.1255 rz=0.1212 rad
          Folder AB
            'desbaste_inicial'
            bajada_broca := p[0,0,-0.012,0,0,0]
            barrenos_menos1 := 8
            barreno_actual := 2
            Loop While (checkContinuously=false) expression=barreno_actual≤barrenos_menos1
              Folder Perforacion
                MoveL speed 100 mm/s, acceleration 500 mm/s^2 (useActiveTCP=true) feature=Base
                  internos := interpolate_pose(Linea1_A, Linea1_B, barreno_actual/barrenos_menos1)
                  Waypoint Waypoint (Variable): variable=internos
                  'desbaste_inicial'
                  bajada_broca := p[0,0,-0.026,0,0,0]
                  bajada := p[0,0,0.026,0,0,0]
                  MoveDirectionNode (selectedDirection=ZMinus toolParams=0.015, 0.015)
                    Until DISTANCE (allowActions=false deceleration=3 distanceNodeType=STOP) Distance=0.0827; motionParameters(blendRadius=0)
                  Popup Message (haltProgram=false message=punto contacto alanzdo inputType=Text)
                  MoveDirectionNode (selectedDirection=ZPlus toolParams=0.003, 0.005)
                    Until DISTANCE (allowActions=false deceleration=3 distanceNodeType=STOP) Distance=0.002; motionParameters(blendRadius=0)
                  Wait Sleep waitTime=0.3
                  Set DigitalOutput pin=config_out[1]; digitalValue=1
                  Wait Sleep waitTime=0.3
                  Loop Counting (count=1) loopVariable(name=Loop_82)
                    bajar := pose_add(get_actual_tcp_pose(), bajada_broca)
                    Waypoint Waypoint (Variable): motionParameters(jointSpeed=1.047198 jointAcceleration=1.396263 cartesianSpeed=0.001 cartesianAcceleration=0.005); variable=bajar
                    subir := pose_sub(get_actual_tcp_pose(), bajada_broca)
                    Waypoint Waypoint (Variable): motionParameters(jointSpeed=1.047198 jointAcceleration=1.396263 cartesianSpeed=0.005 cartesianAcceleration=0.01); variable=subir
                    bajada_broca := pose_sub(bajada_broca, bajada)
                  MoveDirectionNode (selectedDirection=ZPlus toolParams=0.03, 0.035)
                    Until DISTANCE (allowActions=false deceleration=3 distanceNodeType=STOP) Distance=0.06; motionParameters(blendRadius=0)
                  Set DigitalOutput pin=config_out[1]; digitalValue=0
                  barreno_actual := barreno_actual+1
                  Call Quitar_broca
                  Call Poner_broca
          Folder CD
            'desbaste_inicial'
            bajada_broca := p[0,0,-0.012,0,0,0]
            barrenos_menos1 := 8
            barreno_actual := 5
            Loop While (checkContinuously=false) expression=barreno_actual≤barrenos_menos1
              Folder Perforacion
                MoveL speed 100 mm/s, acceleration 500 mm/s^2 (useActiveTCP=true) feature=Base
                  internos := interpolate_pose(Linea1_C, Linea1_D, barreno_actual/barrenos_menos1)
                  Waypoint Waypoint (Variable): variable=internos
                  'desbaste_inicial'
                  bajada_broca := p[0,0,-0.026,0,0,0]
                  bajada := p[0,0,0.026,0,0,0]
                  MoveDirectionNode (selectedDirection=ZMinus toolParams=0.015, 0.015)
                    Until DISTANCE (allowActions=false deceleration=3 distanceNodeType=STOP) Distance=0.0827; motionParameters(blendRadius=0)
                  Popup Message (haltProgram=false message=punto contacto alanzdo inputType=Text)
                  MoveDirectionNode (selectedDirection=ZPlus toolParams=0.003, 0.005)
                    Until DISTANCE (allowActions=false deceleration=3 distanceNodeType=STOP) Distance=0.002; motionParameters(blendRadius=0)
                  Wait Sleep waitTime=0.3
                  Set DigitalOutput pin=config_out[1]; digitalValue=1
                  Wait Sleep waitTime=0.3
                  Loop Counting (count=1) loopVariable(name=Loop_85)
                    bajar := pose_add(get_actual_tcp_pose(), bajada_broca)
                    Waypoint Waypoint (Variable): motionParameters(jointSpeed=1.047198 jointAcceleration=1.396263 cartesianSpeed=0.001 cartesianAcceleration=0.005); variable=bajar
                    subir := pose_sub(get_actual_tcp_pose(), bajada_broca)
                    Waypoint Waypoint (Variable): motionParameters(jointSpeed=1.047198 jointAcceleration=1.396263 cartesianSpeed=0.005 cartesianAcceleration=0.01); variable=subir
                    bajada_broca := pose_sub(bajada_broca, bajada)
                  MoveDirectionNode (selectedDirection=ZPlus toolParams=0.03, 0.035)
                    Until DISTANCE (allowActions=false deceleration=3 distanceNodeType=STOP) Distance=0.06; motionParameters(blendRadius=0)
                  Set DigitalOutput pin=config_out[1]; digitalValue=0
                  barreno_actual := barreno_actual+1
                  Call Quitar_broca
                  Call Poner_broca
          Folder EF
            'desbaste_inicial'
            bajada_broca := p[0,0,-0.012,0,0,0]
            barrenos_menos1 := 8
            barreno_actual := 0
            Loop While (checkContinuously=false) expression=barreno_actual≤barrenos_menos1
              Folder Perforacion
                MoveL speed 100 mm/s, acceleration 500 mm/s^2 (useActiveTCP=true) feature=Base
                  internos := interpolate_pose(Linea1_E, Linea1_F, barreno_actual/barrenos_menos1)
                  Waypoint Waypoint (Variable): variable=internos
                  'desbaste_inicial'
                  bajada_broca := p[0,0,-0.026,0,0,0]
                  bajada := p[0,0,0.026,0,0,0]
                  MoveDirectionNode (selectedDirection=ZMinus toolParams=0.015, 0.015)
                    Until DISTANCE (allowActions=false deceleration=3 distanceNodeType=STOP) Distance=0.0827; motionParameters(blendRadius=0)
                  Popup Message (haltProgram=false message=punto contacto alanzdo inputType=Text)
                  MoveDirectionNode (selectedDirection=ZPlus toolParams=0.003, 0.005)
                    Until DISTANCE (allowActions=false deceleration=3 distanceNodeType=STOP) Distance=0.002; motionParameters(blendRadius=0)
                  Wait Sleep waitTime=0.3
                  Set DigitalOutput pin=config_out[1]; digitalValue=1
                  Wait Sleep waitTime=0.3
                  Loop Counting (count=1) loopVariable(name=Loop_87)
                    bajar := pose_add(get_actual_tcp_pose(), bajada_broca)
                    Waypoint Waypoint (Variable): motionParameters(jointSpeed=1.047198 jointAcceleration=1.396263 cartesianSpeed=0.001 cartesianAcceleration=0.005); variable=bajar
                    subir := pose_sub(get_actual_tcp_pose(), bajada_broca)
                    Waypoint Waypoint (Variable): motionParameters(jointSpeed=1.047198 jointAcceleration=1.396263 cartesianSpeed=0.005 cartesianAcceleration=0.01); variable=subir
                    bajada_broca := pose_sub(bajada_broca, bajada)
                  MoveDirectionNode (selectedDirection=ZPlus toolParams=0.03, 0.035)
                    Until DISTANCE (allowActions=false deceleration=3 distanceNodeType=STOP) Distance=0.06; motionParameters(blendRadius=0)
                  Set DigitalOutput pin=config_out[1]; digitalValue=0
                  barreno_actual := barreno_actual+1
                  Call Quitar_broca
                  Call Poner_broca
        Popup Message (haltProgram=false message=Linea1 con full Terminada! inputType=Text)
        Folder Linea2
          Folder Marcar_puntos
            MoveL speed 100 mm/s, acceleration 500 mm/s^2 (useActiveTCP=true) feature=Base
              Waypoint Home2: TCP in base x=649.602 y=3.2 z=254.15 mm, rx=-2.4485 ry=-1.9662 rz=-0.0111 rad; joints [-199.372, -96.579, 116.673, -19.801, -286.041, 0.348] deg; TCP offset x=0.411 y=-218.298 z=37.994 mm, rx=1.558 ry=-0.1255 rz=0.1212 rad
              Waypoint Linea2_A: TCP in base x=466.954 y=182.157 z=110.172 mm, rx=-2.4485 ry=-1.9662 rz=-0.0111 rad; joints [-177.403, -103.734, 138.62, -34.639, -264.097, 0.47] deg; TCP offset x=0.411 y=-218.298 z=37.994 mm, rx=1.558 ry=-0.1255 rz=0.1212 rad
              Waypoint Linea2_B: TCP in base x=671.81 y=182.878 z=110.175 mm, rx=-2.4484 ry=-1.9662 rz=-0.011 rad; joints [-178.316, -83.76, 120.353, -36.338, -265.022, 0.484] deg; TCP offset x=0.411 y=-218.298 z=37.994 mm, rx=1.558 ry=-0.1255 rz=0.1212 rad
              Waypoint Linea2_C: TCP in base x=694.981 y=182.77 z=110.46 mm, rx=-2.4483 ry=-1.9662 rz=-0.0109 rad; joints [-178.397, -81.801, 118.029, -35.97, -265.106, 0.486] deg; TCP offset x=0.411 y=-218.298 z=37.994 mm, rx=1.558 ry=-0.1255 rz=0.1212 rad
              Waypoint Linea2_D: TCP in base x=898.787 y=183.235 z=110.403 mm, rx=-2.4483 ry=-1.9664 rz=-0.011 rad; joints [-178.787, -65.181, 95.382, -29.948, -265.491, 0.487] deg
              Waypoint Linea2_E: TCP in base x=923.79 y=182.507 z=110.324 mm, rx=-2.4483 ry=-1.9664 rz=-0.011 rad; joints [-178.879, -63.164, 92.292, -28.877, -265.58, 0.486] deg
              Waypoint Linea2_F: TCP in base x=1126.946 y=182.371 z=110.084 mm, rx=-2.4483 ry=-1.9664 rz=-0.011 rad; joints [-179.118, -45.199, 62.135, -16.683, -265.793, 0.483] deg
          Folder AB
            'desbaste_inicial'
            bajada_broca := p[0,0,-0.012,0,0,0]
            barrenos_menos1 := 8
            barreno_actual := 0
            Loop While (checkContinuously=false) expression=barreno_actual≤barrenos_menos1
              Folder Perforacion
                MoveL speed 100 mm/s, acceleration 500 mm/s^2 (useActiveTCP=true) feature=Base
                  internos := interpolate_pose(Linea2_A, Linea2_B, barreno_actual/barrenos_menos1)
                  Waypoint Waypoint (Variable): variable=internos
                  'desbaste_inicial'
                  bajada_broca := p[0,0,-0.026,0,0,0]
                  bajada := p[0,0,0.026,0,0,0]
                  MoveDirectionNode (selectedDirection=ZMinus toolParams=0.015, 0.015)
                    Until DISTANCE (allowActions=false deceleration=3 distanceNodeType=STOP) Distance=0.0827; motionParameters(blendRadius=0)
                  Popup Message (haltProgram=false message=punto contacto alanzdo inputType=Text)
                  MoveDirectionNode (selectedDirection=ZPlus toolParams=0.003, 0.005)
                    Until DISTANCE (allowActions=false deceleration=3 distanceNodeType=STOP) Distance=0.002; motionParameters(blendRadius=0)
                  Wait Sleep waitTime=0.3
                  Set DigitalOutput pin=config_out[1]; digitalValue=1
                  Wait Sleep waitTime=0.3
                  Loop Counting (count=1) loopVariable(name=Loop_90)
                    bajar := pose_add(get_actual_tcp_pose(), bajada_broca)
                    Waypoint Waypoint (Variable): motionParameters(jointSpeed=1.047198 jointAcceleration=1.396263 cartesianSpeed=0.001 cartesianAcceleration=0.005); variable=bajar
                    subir := pose_sub(get_actual_tcp_pose(), bajada_broca)
                    Waypoint Waypoint (Variable): motionParameters(jointSpeed=1.047198 jointAcceleration=1.396263 cartesianSpeed=0.005 cartesianAcceleration=0.01); variable=subir
                    bajada_broca := pose_sub(bajada_broca, bajada)
                  MoveDirectionNode (selectedDirection=ZPlus toolParams=0.03, 0.035)
                    Until DISTANCE (allowActions=false deceleration=3 distanceNodeType=STOP) Distance=0.06; motionParameters(blendRadius=0)
                  Set DigitalOutput pin=config_out[1]; digitalValue=0
                  barreno_actual := barreno_actual+1
                  Call Quitar_broca
                  Call Poner_broca
          Folder CD
            'desbaste_inicial'
            bajada_broca := p[0,0,-0.012,0,0,0]
            barrenos_menos1 := 8
            barreno_actual := 0
            Loop While (checkContinuously=false) expression=barreno_actual≤barrenos_menos1
              Folder Perforacion
                MoveL speed 100 mm/s, acceleration 500 mm/s^2 (useActiveTCP=true) feature=Base
                  internos := interpolate_pose(Linea2_C, Linea2_D, barreno_actual/barrenos_menos1)
                  Waypoint Waypoint (Variable): variable=internos
                  'desbaste_inicial'
                  bajada_broca := p[0,0,-0.026,0,0,0]
                  bajada := p[0,0,0.026,0,0,0]
                  MoveDirectionNode (selectedDirection=ZMinus toolParams=0.015, 0.015)
                    Until DISTANCE (allowActions=false deceleration=3 distanceNodeType=STOP) Distance=0.0827; motionParameters(blendRadius=0)
                  Popup Message (haltProgram=false message=punto contacto alanzdo inputType=Text)
                  MoveDirectionNode (selectedDirection=ZPlus toolParams=0.003, 0.005)
                    Until DISTANCE (allowActions=false deceleration=3 distanceNodeType=STOP) Distance=0.002; motionParameters(blendRadius=0)
                  Wait Sleep waitTime=0.3
                  Set DigitalOutput pin=config_out[1]; digitalValue=1
                  Wait Sleep waitTime=0.3
                  Loop Counting (count=1) loopVariable(name=Loop_92)
                    bajar := pose_add(get_actual_tcp_pose(), bajada_broca)
                    Waypoint Waypoint (Variable): motionParameters(jointSpeed=1.047198 jointAcceleration=1.396263 cartesianSpeed=0.001 cartesianAcceleration=0.005); variable=bajar
                    subir := pose_sub(get_actual_tcp_pose(), bajada_broca)
                    Waypoint Waypoint (Variable): motionParameters(jointSpeed=1.047198 jointAcceleration=1.396263 cartesianSpeed=0.005 cartesianAcceleration=0.01); variable=subir
                    bajada_broca := pose_sub(bajada_broca, bajada)
                  MoveDirectionNode (selectedDirection=ZPlus toolParams=0.03, 0.035)
                    Until DISTANCE (allowActions=false deceleration=3 distanceNodeType=STOP) Distance=0.06; motionParameters(blendRadius=0)
                  Set DigitalOutput pin=config_out[1]; digitalValue=0
                  barreno_actual := barreno_actual+1
                  Call Quitar_broca
                  Call Poner_broca
          Folder EF
            'desbaste_inicial'
            bajada_broca := p[0,0,-0.012,0,0,0]
            barrenos_menos1 := 8
            barreno_actual := 0
            Loop While (checkContinuously=false) expression=barreno_actual≤barrenos_menos1
              Folder Perforacion
                MoveL speed 100 mm/s, acceleration 500 mm/s^2 (useActiveTCP=true) feature=Base
                  internos := interpolate_pose(Linea2_E, Linea2_F, barreno_actual/barrenos_menos1)
                  Waypoint Waypoint (Variable): variable=internos
                  'desbaste_inicial'
                  bajada_broca := p[0,0,-0.026,0,0,0]
                  bajada := p[0,0,0.026,0,0,0]
                  MoveDirectionNode (selectedDirection=ZMinus toolParams=0.015, 0.015)
                    Until DISTANCE (allowActions=false deceleration=3 distanceNodeType=STOP) Distance=0.0827; motionParameters(blendRadius=0)
                  Popup Message (haltProgram=false message=punto contacto alanzdo inputType=Text)
                  MoveDirectionNode (selectedDirection=ZPlus toolParams=0.003, 0.005)
                    Until DISTANCE (allowActions=false deceleration=3 distanceNodeType=STOP) Distance=0.002; motionParameters(blendRadius=0)
                  Wait Sleep waitTime=0.3
                  Set DigitalOutput pin=config_out[1]; digitalValue=1
                  Wait Sleep waitTime=0.3
                  Loop Counting (count=1) loopVariable(name=Loop_94)
                    bajar := pose_add(get_actual_tcp_pose(), bajada_broca)
                    Waypoint Waypoint (Variable): motionParameters(jointSpeed=1.047198 jointAcceleration=1.396263 cartesianSpeed=0.001 cartesianAcceleration=0.005); variable=bajar
                    subir := pose_sub(get_actual_tcp_pose(), bajada_broca)
                    Waypoint Waypoint (Variable): motionParameters(jointSpeed=1.047198 jointAcceleration=1.396263 cartesianSpeed=0.005 cartesianAcceleration=0.01); variable=subir
                    bajada_broca := pose_sub(bajada_broca, bajada)
                  MoveDirectionNode (selectedDirection=ZPlus toolParams=0.03, 0.035)
                    Until DISTANCE (allowActions=false deceleration=3 distanceNodeType=STOP) Distance=0.06; motionParameters(blendRadius=0)
                  Set DigitalOutput pin=config_out[1]; digitalValue=0
                  barreno_actual := barreno_actual+1
                  If barreno_actual≥barrenos_menos1
                    cambiar_broca := True
                  Call Quitar_broca
                  Call Poner_broca
        Popup Message (haltProgram=false message=Linea2 con full Terminada! inputType=Text)
    Folder 600
      SuppressedNode
        Folder Broca_1
          Folder Linea7
            Folder Marcar_puntos
              MoveL speed 100 mm/s, acceleration 500 mm/s^2 (useActiveTCP=true) feature=Base
                Waypoint Home2: TCP in base x=-476.229 y=0 z=568.737 mm, rx=2.0263 ry=-2.3929 rz=-0.0208 rad; joints [-32.551, -116.469, 98.413, 17.843, -302.102, -0.163] deg; TCP offset x=0.411 y=-218.298 z=37.994 mm, rx=1.558 ry=-0.1255 rz=0.1212 rad
                Waypoint Linea7_A: TCP in base x=737.913 y=-359.697 z=110.247 mm, rx=3.1319 ry=0.1866 rz=-0.0004 rad; joints [-210.915, -68.733, 100.688, -31.639, -226.901, 0.305] deg; TCP offset x=0.411 y=-218.298 z=37.994 mm, rx=1.558 ry=-0.1255 rz=0.1212 rad
                Waypoint Linea7_B: TCP in base x=783.713 y=-360.081 z=110.621 mm, rx=3.1319 ry=0.1866 rz=-0.0004 rad; joints [-209.138, -65.085, 95.206, -29.798, -225.12, 0.318] deg
            Folder AB
              'desbaste_inicial'
              bajada_broca := p[0,0,-0.008,0,0,0]
              barrenos_menos1 := 2
              barreno_actual := 0
              Loop While (checkContinuously=false) expression=barreno_actual≤barrenos_menos1
                Folder Perforacion
                  MoveL speed 100 mm/s, acceleration 500 mm/s^2 (useActiveTCP=true) feature=Base
                    internos := interpolate_pose(Linea7_A, Linea7_B, barreno_actual/barrenos_menos1)
                    Waypoint Waypoint (Variable): variable=internos
                    'desbaste_inicial'
                    bajada_broca := p[0,0,-0.024,0,0,0]
                    bajada := p[0,0,0.024,0,0,0]
                    MoveDirectionNode (selectedDirection=ZMinus toolParams=0.1, 0.15)
                      Until DISTANCE (allowActions=false deceleration=3 distanceNodeType=STOP) Distance=0.071; motionParameters(blendRadius=0)
                    MoveDirectionNode (selectedDirection=ZMinus toolParams=0.01, 0.01)
                      Until TOOL_CONTACT_DETECTION (allowActions=false retraction=0 decelerationAcceleration=0.01 decelerationAngularAcceleration=34.906585)
                    Popup Message (haltProgram=false message=punto contacto alanzdo inputType=Text)
                    MoveDirectionNode (selectedDirection=ZPlus toolParams=0.003, 0.005)
                      Until DISTANCE (allowActions=false deceleration=3 distanceNodeType=STOP) Distance=0.002; motionParameters(blendRadius=0)
                    Wait Sleep waitTime=0.3
                    Set DigitalOutput pin=config_out[1]; digitalValue=1
                    Wait Sleep waitTime=0.3
                    Loop Counting (count=1) loopVariable=Loop_56
                      bajar := pose_add(get_actual_tcp_pose(), bajada_broca)
                      Waypoint Waypoint (Variable): motionParameters(jointSpeed=1.047198 jointAcceleration=1.396263 cartesianSpeed=0.001 cartesianAcceleration=0.005); variable=bajar
                      subir := pose_sub(get_actual_tcp_pose(), bajada_broca)
                      Waypoint Waypoint (Variable): motionParameters(jointSpeed=1.047198 jointAcceleration=1.396263 cartesianSpeed=0.005 cartesianAcceleration=0.01); variable=subir
                      bajada_broca := pose_sub(bajada_broca, bajada)
                    MoveDirectionNode (selectedDirection=ZPlus toolParams=0.1, 0.15)
                      Until DISTANCE (allowActions=false deceleration=3 distanceNodeType=STOP) Distance=0.08; motionParameters(blendRadius=0)
                    Set DigitalOutput pin=config_out[1]; digitalValue=0
                    barreno_actual := barreno_actual+1
                    Call Quitar_broca
                    Call Poner_broca
          Popup Message (haltProgram=false message=Linea7 con chica Terminada! inputType=Text)
          Folder Linea8
            Folder Marcar_puntos
              MoveL speed 100 mm/s, acceleration 500 mm/s^2 (useActiveTCP=true) feature=Base
                Waypoint Linea8_A: TCP in base x=886.283 y=-360.229 z=110.454 mm, rx=3.1315 ry=0.1865 rz=0.0006 rad; joints [-205.767, -56.675, 81.874, -24.901, -221.735, 0.344] deg
                Waypoint Linea8_B: TCP in base x=1009.987 y=-360.229 z=110.179 mm, rx=3.1315 ry=0.1865 rz=0.0006 rad; joints [-202.59, -45.403, 62.493, -16.778, -218.539, 0.367] deg
            Folder AB
              'desbaste_inicial'
              bajada_broca := p[0,0,-0.008,0,0,0]
              barrenos_menos1 := 5
              barreno_actual := 0
              Loop While (checkContinuously=false) expression=barreno_actual≤barrenos_menos1
                Folder Perforacion
                  MoveL speed 100 mm/s, acceleration 500 mm/s^2 (useActiveTCP=true) feature=Base
                    internos := interpolate_pose(Linea8_A, Linea8_B, barreno_actual/barrenos_menos1)
                    Waypoint Waypoint (Variable): variable=internos
                    'desbaste_inicial'
                    bajada_broca := p[0,0,-0.008,0,0,0]
                    bajada := p[0,0,0.008,0,0,0]
                    MoveDirectionNode (selectedDirection=ZMinus toolParams=0.1, 0.15)
                      Until DISTANCE (allowActions=false deceleration=3 distanceNodeType=STOP) Distance=0.071; motionParameters(blendRadius=0)
                    MoveDirectionNode (selectedDirection=ZMinus toolParams=0.01, 0.01)
                      Until TOOL_CONTACT_DETECTION (allowActions=false retraction=0 decelerationAcceleration=0.01 decelerationAngularAcceleration=34.906585)
                    Popup Message (haltProgram=false message=punto contacto alanzdo inputType=Text)
                    MoveDirectionNode (selectedDirection=ZPlus toolParams=0.003, 0.005)
                      Until DISTANCE (allowActions=false deceleration=3 distanceNodeType=STOP) Distance=0.002; motionParameters(blendRadius=0)
                    Wait Sleep waitTime=0.3
                    Set DigitalOutput pin=config_out[1]; digitalValue=1
                    Wait Sleep waitTime=0.3
                    SuppressedNode
                      Loop Counting (count=3) loopVariable(name=Loop_68)
                        bajar := pose_add(get_actual_tcp_pose(), bajada_broca)
                        Waypoint Waypoint (Variable): motionParameters(jointSpeed=1.047198 jointAcceleration=1.396263 cartesianSpeed=0.001 cartesianAcceleration=0.005); variable=bajar
                        subir := pose_sub(get_actual_tcp_pose(), bajada_broca)
                        Waypoint Waypoint (Variable): motionParameters(jointSpeed=1.047198 jointAcceleration=1.396263 cartesianSpeed=0.005 cartesianAcceleration=0.01); variable=subir
                        bajada_broca := pose_sub(bajada_broca, bajada)
                    MoveDirectionNode (selectedDirection=ZPlus toolParams=0.1, 0.15)
                      Until DISTANCE (allowActions=false deceleration=3 distanceNodeType=STOP) Distance=0.08; motionParameters(blendRadius=0)
                    Set DigitalOutput pin=config_out[1]; digitalValue=0
                    barreno_actual := barreno_actual+1
                    SuppressedNode
                      Call Quitar_broca
                    SuppressedNode
                      Call Poner_broca
          Popup Message (haltProgram=false message=Linea8 con chica Terminada! inputType=Text)
          Folder Linea9
            Folder Marcar_puntos
              MoveL speed 100 mm/s, acceleration 500 mm/s^2 (useActiveTCP=true) feature=Base
                Waypoint Linea9_A: TCP in base x=1089.313 y=-360.631 z=110.237 mm, rx=3.1313 ry=0.1866 rz=0.0014 rad; joints [-200.952, -36.589, 46.349, -9.474, -216.885, 0.379] deg
                Waypoint Linea9_B: TCP in base x=1138.944 y=-360.869 z=110.826 mm, rx=3.1313 ry=0.1866 rz=0.0014 rad; joints [-200.044, -29.362, 32.524, -2.871, -215.958, 0.386] deg
            Folder AB
              'desbaste_inicial'
              bajada_broca := p[0,0,-0.008,0,0,0]
              barrenos_menos1 := 2
              barreno_actual := 0
              Loop While (checkContinuously=false) expression=barreno_actual≤barrenos_menos1
                Folder Perforacion
                  MoveL speed 100 mm/s, acceleration 500 mm/s^2 (useActiveTCP=true) feature=Base
                    internos := interpolate_pose(Linea9_A, Linea9_B, barreno_actual/barrenos_menos1)
                    Waypoint Waypoint (Variable): variable=internos
                    'desbaste_inicial'
                    bajada_broca := p[0,0,-0.008,0,0,0]
                    bajada := p[0,0,0.008,0,0,0]
                    MoveDirectionNode (selectedDirection=ZMinus toolParams=0.1, 0.15)
                      Until DISTANCE (allowActions=false deceleration=3 distanceNodeType=STOP) Distance=0.071; motionParameters(blendRadius=0)
                    MoveDirectionNode (selectedDirection=ZMinus toolParams=0.01, 0.01)
                      Until TOOL_CONTACT_DETECTION (allowActions=false retraction=0 decelerationAcceleration=0.01 decelerationAngularAcceleration=34.906585)
                    Popup Message (haltProgram=false message=punto contacto alanzdo inputType=Text)
                    MoveDirectionNode (selectedDirection=ZPlus toolParams=0.003, 0.005)
                      Until DISTANCE (allowActions=false deceleration=3 distanceNodeType=STOP) Distance=0.002; motionParameters(blendRadius=0)
                    Wait Sleep waitTime=0.3
                    Set DigitalOutput pin=config_out[1]; digitalValue=1
                    Wait Sleep waitTime=0.3
                    SuppressedNode
                      Loop Counting (count=3) loopVariable(name=Loop_74)
                        bajar := pose_add(get_actual_tcp_pose(), bajada_broca)
                        Waypoint Waypoint (Variable): motionParameters(jointSpeed=1.047198 jointAcceleration=1.396263 cartesianSpeed=0.001 cartesianAcceleration=0.005); variable=bajar
                        subir := pose_sub(get_actual_tcp_pose(), bajada_broca)
                        Waypoint Waypoint (Variable): motionParameters(jointSpeed=1.047198 jointAcceleration=1.396263 cartesianSpeed=0.005 cartesianAcceleration=0.01); variable=subir
                        bajada_broca := pose_sub(bajada_broca, bajada)
                    MoveDirectionNode (selectedDirection=ZPlus toolParams=0.1, 0.15)
                      Until DISTANCE (allowActions=false deceleration=3 distanceNodeType=STOP) Distance=0.08; motionParameters(blendRadius=0)
                    Set DigitalOutput pin=config_out[1]; digitalValue=0
                    barreno_actual := barreno_actual+1
                    SuppressedNode
                      Call Quitar_broca
                    SuppressedNode
                      Call Poner_broca
          Popup Message (haltProgram=false message=Linea9 con chica Terminada! inputType=Text)
          Folder Linea10
            Folder Marcar_puntos
              MoveL speed 100 mm/s, acceleration 500 mm/s^2 (useActiveTCP=true) feature=Base
                Waypoint Home2: TCP in base x=-476.229 y=0 z=568.737 mm, rx=2.0263 ry=-2.3929 rz=-0.0208 rad; joints [-32.551, -116.469, 98.413, 17.843, -302.102, -0.163] deg; TCP offset x=0.411 y=-218.298 z=37.994 mm, rx=1.558 ry=-0.1255 rz=0.1212 rad
                Waypoint Linea10_A: TCP in base x=620.978 y=-324.892 z=110.624 mm, rx=3.1274 ry=-0.2451 rz=-0.0041 rad; joints [-211.246, -75.766, 110.43, -34.284, -211.451, 0.322] deg; TCP offset x=0.411 y=-218.298 z=37.994 mm, rx=1.558 ry=-0.1255 rz=0.1212 rad
                Waypoint Linea10_B: TCP in base x=621.098 y=-276.98 z=110.32 mm, rx=3.1274 ry=-0.2451 rz=-0.0041 rad; joints [-207.342, -76.685, 111.673, -34.563, -207.548, 0.378] deg
            Folder AB
              'desbaste_inicial'
              bajada_broca := p[0,0,-0.008,0,0,0]
              barrenos_menos1 := 2
              barreno_actual := 0
              Loop While (checkContinuously=false) expression=barreno_actual≤barrenos_menos1
                Folder Perforacion
                  MoveL speed 100 mm/s, acceleration 500 mm/s^2 (useActiveTCP=true) feature=Base
                    internos := interpolate_pose(Linea10_A, Linea10_B, barreno_actual/barrenos_menos1)
                    Waypoint Waypoint (Variable): variable=internos
                    'desbaste_inicial'
                    bajada_broca := p[0,0,-0.008,0,0,0]
                    bajada := p[0,0,0.008,0,0,0]
                    MoveDirectionNode (selectedDirection=ZMinus toolParams=0.1, 0.15)
                      Until DISTANCE (allowActions=false deceleration=3 distanceNodeType=STOP) Distance=0.071; motionParameters(blendRadius=0)
                    MoveDirectionNode (selectedDirection=ZMinus toolParams=0.001, 0.001)
                      Until TOOL_CONTACT_DETECTION (allowActions=false retraction=0 decelerationAcceleration=0.001 decelerationAngularAcceleration=34.906585)
                    Popup Message (haltProgram=false message=punto contacto alanzdo inputType=Text)
                    MoveDirectionNode (selectedDirection=ZPlus toolParams=0.003, 0.005)
                      Until DISTANCE (allowActions=false deceleration=3 distanceNodeType=STOP) Distance=0.002; motionParameters(blendRadius=0)
                    Wait Sleep waitTime=0.3
                    Set DigitalOutput pin=config_out[1]; digitalValue=1
                    Wait Sleep waitTime=0.3
                    SuppressedNode
                      Loop Counting (count=3) loopVariable(name=Loop_76)
                        bajar := pose_add(get_actual_tcp_pose(), bajada_broca)
                        Waypoint Waypoint (Variable): motionParameters(jointSpeed=1.047198 jointAcceleration=1.396263 cartesianSpeed=0.001 cartesianAcceleration=0.005); variable=bajar
                        subir := pose_sub(get_actual_tcp_pose(), bajada_broca)
                        Waypoint Waypoint (Variable): motionParameters(jointSpeed=1.047198 jointAcceleration=1.396263 cartesianSpeed=0.005 cartesianAcceleration=0.01); variable=subir
                        bajada_broca := pose_sub(bajada_broca, bajada)
                    MoveDirectionNode (selectedDirection=ZPlus toolParams=0.1, 0.15)
                      Until DISTANCE (allowActions=false deceleration=3 distanceNodeType=STOP) Distance=0.08; motionParameters(blendRadius=0)
                    Set DigitalOutput pin=config_out[1]; digitalValue=0
                    barreno_actual := barreno_actual+1
                    SuppressedNode
                      Call Quitar_broca
                    SuppressedNode
                      Call Poner_broca
          Popup Message (haltProgram=false message=Linea10 con chica Terminada! inputType=Text)
          Folder Linea11
            Folder Marcar_puntos
              MoveL speed 100 mm/s, acceleration 500 mm/s^2 (useActiveTCP=true) feature=Base
                Waypoint Linea11_A: TCP in base x=-636.133 y=-137.915 z=110.44 mm, rx=2.0204 ry=-2.394 rz=-0.0205 rad; joints [-4.201, -88.707, 125.915, -37.584, -273.698, -0.078] deg; TCP offset x=0.411 y=-218.298 z=37.994 mm, rx=1.558 ry=-0.1255 rz=0.1212 rad
                Waypoint Linea11_B: TCP in base x=-635.407 y=-82.609 z=110.403 mm, rx=2.0204 ry=-2.3939 rz=-0.0206 rad; joints [-11.006, -90.015, 127.249, -37.609, -280.504, -0.032] deg
            Folder AB
              'desbaste_inicial'
              bajada_broca := p[0,0,-0.008,0,0,0]
              barrenos_menos1 := 2
              barreno_actual := 0
              Loop While (checkContinuously=false) expression=barreno_actual≤barrenos_menos1
                Folder Perforacion
                  MoveL speed 100 mm/s, acceleration 500 mm/s^2 (useActiveTCP=true) feature=Base
                    SuppressedNode
                      If barreno_actual≟5
                        barreno_actual := barreno_actual+1
                    internos := interpolate_pose(Linea11_A, Linea11_B, barreno_actual/barrenos_menos1)
                    Waypoint Waypoint (Variable): variable=internos
                    'desbaste_inicial'
                    bajada_broca := p[0,0,-0.008,0,0,0]
                    bajada := p[0,0,0.008,0,0,0]
                    MoveDirectionNode (selectedDirection=ZMinus toolParams=0.1, 0.15)
                      Until DISTANCE (allowActions=false deceleration=3 distanceNodeType=STOP) Distance=0.071; motionParameters(blendRadius=0)
                    MoveDirectionNode (selectedDirection=ZMinus toolParams=0.001, 0.001)
                      Until TOOL_CONTACT_DETECTION (allowActions=false retraction=0 decelerationAcceleration=0.001 decelerationAngularAcceleration=34.906585)
                    Popup Message (haltProgram=false message=punto contacto alanzdo inputType=Text)
                    MoveDirectionNode (selectedDirection=ZPlus toolParams=0.003, 0.005)
                      Until DISTANCE (allowActions=false deceleration=3 distanceNodeType=STOP) Distance=0.002; motionParameters(blendRadius=0)
                    Wait Sleep waitTime=0.3
                    Set DigitalOutput pin=config_out[1]; digitalValue=1
                    Wait Sleep waitTime=0.3
                    SuppressedNode
                      Loop Counting (count=3) loopVariable=Loop_80
                        bajar := pose_add(get_actual_tcp_pose(), bajada_broca)
                        Waypoint Waypoint (Variable): motionParameters(jointSpeed=1.047198 jointAcceleration=1.396263 cartesianSpeed=0.001 cartesianAcceleration=0.005); variable=bajar
                        subir := pose_sub(get_actual_tcp_pose(), bajada_broca)
                        Waypoint Waypoint (Variable): motionParameters(jointSpeed=1.047198 jointAcceleration=1.396263 cartesianSpeed=0.005 cartesianAcceleration=0.01); variable=subir
                        bajada_broca := pose_sub(bajada_broca, bajada)
                    MoveDirectionNode (selectedDirection=ZPlus toolParams=0.1, 0.15)
                      Until DISTANCE (allowActions=false deceleration=3 distanceNodeType=STOP) Distance=0.08; motionParameters(blendRadius=0)
                    Set DigitalOutput pin=config_out[1]; digitalValue=0
                    barreno_actual := barreno_actual+1
                    SuppressedNode
                      Call Quitar_broca
                    SuppressedNode
                      Call Poner_broca
          Popup Message (haltProgram=false message=Linea11 con chica Terminada! inputType=Text)
          Folder Linea12
            Folder Marcar_puntos
              MoveL speed 100 mm/s, acceleration 500 mm/s^2 (useActiveTCP=true) feature=Base
                Waypoint Linea12_A: TCP in base x=624.141 y=-66.274 z=110.335 mm, rx=-2.6321 ry=-1.7106 rz=-0.0087 rad; joints [-204.939, -91.033, 128.004, -36.559, -280.152, 0.387] deg
                Waypoint Linea12_B: TCP in base x=625.005 y=106.664 z=110.181 mm, rx=-2.6321 ry=-1.7106 rz=-0.0087 rad; joints [-183.741, -88.918, 125.907, -36.601, -258.955, 0.536] deg
            Folder AB
              'desbaste_inicial'
              bajada_broca := p[0,0,-0.008,0,0,0]
              barrenos_menos1 := 7
              barreno_actual := 0
              Loop While (checkContinuously=false) expression=barreno_actual≤barrenos_menos1
                Folder Perforacion
                  MoveL speed 100 mm/s, acceleration 500 mm/s^2 (useActiveTCP=true) feature=Base
                    If barreno_actual≟2
                      barreno_actual := barreno_actual+1
                    internos := interpolate_pose(Linea12_A, Linea12_B, barreno_actual/barrenos_menos1)
                    Waypoint Waypoint (Variable): variable=internos
                    'desbaste_inicial'
                    bajada_broca := p[0,0,-0.008,0,0,0]
                    bajada := p[0,0,0.008,0,0,0]
                    MoveDirectionNode (selectedDirection=ZMinus toolParams=0.1, 0.15)
                      Until DISTANCE (allowActions=false deceleration=3 distanceNodeType=STOP) Distance=0.071; motionParameters(blendRadius=0)
                    MoveDirectionNode (selectedDirection=ZMinus toolParams=0.001, 0.001)
                      Until TOOL_CONTACT_DETECTION (allowActions=false retraction=0 decelerationAcceleration=0.001 decelerationAngularAcceleration=34.906585)
                    Popup Message (haltProgram=false message=punto contacto alanzdo inputType=Text)
                    MoveDirectionNode (selectedDirection=ZPlus toolParams=0.003, 0.005)
                      Until DISTANCE (allowActions=false deceleration=3 distanceNodeType=STOP) Distance=0.002; motionParameters(blendRadius=0)
                    Wait Sleep waitTime=0.3
                    Set DigitalOutput pin=config_out[1]; digitalValue=1
                    Wait Sleep waitTime=0.3
                    SuppressedNode
                      Loop Counting (count=3) loopVariable=Loop_78
                        bajar := pose_add(get_actual_tcp_pose(), bajada_broca)
                        Waypoint Waypoint (Variable): motionParameters(jointSpeed=1.047198 jointAcceleration=1.396263 cartesianSpeed=0.001 cartesianAcceleration=0.005); variable=bajar
                        subir := pose_sub(get_actual_tcp_pose(), bajada_broca)
                        Waypoint Waypoint (Variable): motionParameters(jointSpeed=1.047198 jointAcceleration=1.396263 cartesianSpeed=0.005 cartesianAcceleration=0.01); variable=subir
                        bajada_broca := pose_sub(bajada_broca, bajada)
                    MoveDirectionNode (selectedDirection=ZPlus toolParams=0.1, 0.15)
                      Until DISTANCE (allowActions=false deceleration=3 distanceNodeType=STOP) Distance=0.08; motionParameters(blendRadius=0)
                    Set DigitalOutput pin=config_out[1]; digitalValue=0
                    barreno_actual := barreno_actual+1
                    SuppressedNode
                      Call Quitar_broca
                    SuppressedNode
                      Call Poner_broca
          Popup Message (haltProgram=false message=Linea12 con chica Terminada! inputType=Text)
          Folder Linea13
            Folder Marcar_puntos
              MoveL speed 100 mm/s, acceleration 500 mm/s^2 (useActiveTCP=true) feature=Base
                Waypoint Linea13_A: TCP in base x=625.493 y=262.479 z=110.355 mm, rx=-2.6325 ry=-1.7109 rz=-0.0101 rad; joints [-165.949, -82.781, 119.173, -36.043, -241.164, 0.656] deg
                Waypoint Linea13_B: TCP in base x=625.493 y=318.857 z=110.132 mm, rx=-2.6325 ry=-1.7109 rz=-0.0101 rad; joints [-160.355, -79.919, 115.767, -35.483, -235.569, 0.699] deg
            Folder AB
              'desbaste_inicial'
              bajada_broca := p[0,0,-0.008,0,0,0]
              barrenos_menos1 := 2
              barreno_actual := 0
              Loop While (checkContinuously=false) expression=barreno_actual≤barrenos_menos1
                Folder Perforacion
                  MoveL speed 100 mm/s, acceleration 500 mm/s^2 (useActiveTCP=true) feature=Base
                    SuppressedNode
                      If barreno_actual≟2
                        barreno_actual := barreno_actual+1
                    internos := interpolate_pose(Linea13_A, Linea13_B, barreno_actual/barrenos_menos1)
                    Waypoint Waypoint (Variable): variable=internos
                    'desbaste_inicial'
                    bajada_broca := p[0,0,-0.008,0,0,0]
                    bajada := p[0,0,0.008,0,0,0]
                    MoveDirectionNode (selectedDirection=ZMinus toolParams=0.1, 0.15)
                      Until DISTANCE (allowActions=false deceleration=3 distanceNodeType=STOP) Distance=0.071; motionParameters(blendRadius=0)
                    MoveDirectionNode (selectedDirection=ZMinus toolParams=0.001, 0.001)
                      Until TOOL_CONTACT_DETECTION (allowActions=false retraction=0 decelerationAcceleration=0.001 decelerationAngularAcceleration=34.906585)
                    Popup Message (haltProgram=false message=punto contacto alanzdo inputType=Text)
                    MoveDirectionNode (selectedDirection=ZPlus toolParams=0.003, 0.005)
                      Until DISTANCE (allowActions=false deceleration=3 distanceNodeType=STOP) Distance=0.002; motionParameters(blendRadius=0)
                    Wait Sleep waitTime=0.3
                    Set DigitalOutput pin=config_out[1]; digitalValue=1
                    Wait Sleep waitTime=0.3
                    SuppressedNode
                      Loop Counting (count=3) loopVariable=Loop_82
                        bajar := pose_add(get_actual_tcp_pose(), bajada_broca)
                        Waypoint Waypoint (Variable): motionParameters(jointSpeed=1.047198 jointAcceleration=1.396263 cartesianSpeed=0.001 cartesianAcceleration=0.005); variable=bajar
                        subir := pose_sub(get_actual_tcp_pose(), bajada_broca)
                        Waypoint Waypoint (Variable): motionParameters(jointSpeed=1.047198 jointAcceleration=1.396263 cartesianSpeed=0.005 cartesianAcceleration=0.01); variable=subir
                        bajada_broca := pose_sub(bajada_broca, bajada)
                    MoveDirectionNode (selectedDirection=ZPlus toolParams=0.1, 0.15)
                      Until DISTANCE (allowActions=false deceleration=3 distanceNodeType=STOP) Distance=0.08; motionParameters(blendRadius=0)
                    Set DigitalOutput pin=config_out[1]; digitalValue=0
                    barreno_actual := barreno_actual+1
                    SuppressedNode
                      Call Quitar_broca
                    SuppressedNode
                      Call Poner_broca
          Popup Message (haltProgram=false message=Linea13 con chica Terminada! inputType=Text)
          Folder Linea14
            Folder Marcar_puntos
              MoveL speed 100 mm/s, acceleration 500 mm/s^2 (useActiveTCP=true) feature=Base
                Waypoint Linea14_A: TCP in base x=625.749 y=343.505 z=110.091 mm, rx=-2.6326 ry=-1.7111 rz=-0.011 rad; joints [-158.078, -78.594, 114.13, -35.197, -233.295, 0.717] deg
                Waypoint Linea14_B: TCP in base x=-633.711 y=492.58 z=110.745 mm, rx=2.0205 ry=-2.3939 rz=-0.0205 rad; joints [-60.426, -72.306, 105.929, -34.278, -329.923, 0.504] deg; TCP offset x=0.411 y=-218.298 z=37.994 mm, rx=1.558 ry=-0.1255 rz=0.1212 rad
            Folder AB
              'desbaste_inicial'
              bajada_broca := p[0,0,-0.008,0,0,0]
              barrenos_menos1 := 5
              barreno_actual := 0
              Loop While (checkContinuously=false) expression=barreno_actual≤barrenos_menos1
                Folder Perforacion
                  MoveL speed 100 mm/s, acceleration 500 mm/s^2 (useActiveTCP=true) feature=Base
                    If barreno_actual≟3
                      barreno_actual := barreno_actual+1
                    internos := interpolate_pose(Linea14_A, Linea14_B, barreno_actual/barrenos_menos1)
                    Waypoint Waypoint (Variable): variable=internos
                    'desbaste_inicial'
                    bajada_broca := p[0,0,-0.008,0,0,0]
                    bajada := p[0,0,0.008,0,0,0]
                    MoveDirectionNode (selectedDirection=ZMinus toolParams=0.1, 0.15)
                      Until DISTANCE (allowActions=false deceleration=3 distanceNodeType=STOP) Distance=0.071; motionParameters(blendRadius=0)
                    MoveDirectionNode (selectedDirection=ZMinus toolParams=0.001, 0.001)
                      Until TOOL_CONTACT_DETECTION (allowActions=false retraction=0 decelerationAcceleration=0.001 decelerationAngularAcceleration=34.906585)
                    Popup Message (haltProgram=false message=punto contacto alanzdo inputType=Text)
                    MoveDirectionNode (selectedDirection=ZPlus toolParams=0.003, 0.005)
                      Until DISTANCE (allowActions=false deceleration=3 distanceNodeType=STOP) Distance=0.002; motionParameters(blendRadius=0)
                    Wait Sleep waitTime=0.3
                    Set DigitalOutput pin=config_out[1]; digitalValue=1
                    Wait Sleep waitTime=0.3
                    SuppressedNode
                      Loop Counting (count=3) loopVariable(name=Loop_84)
                        bajar := pose_add(get_actual_tcp_pose(), bajada_broca)
                        Waypoint Waypoint (Variable): motionParameters(jointSpeed=1.047198 jointAcceleration=1.396263 cartesianSpeed=0.001 cartesianAcceleration=0.005); variable=bajar
                        subir := pose_sub(get_actual_tcp_pose(), bajada_broca)
                        Waypoint Waypoint (Variable): motionParameters(jointSpeed=1.047198 jointAcceleration=1.396263 cartesianSpeed=0.005 cartesianAcceleration=0.01); variable=subir
                        bajada_broca := pose_sub(bajada_broca, bajada)
                    MoveDirectionNode (selectedDirection=ZPlus toolParams=0.1, 0.15)
                      Until DISTANCE (allowActions=false deceleration=3 distanceNodeType=STOP) Distance=0.08; motionParameters(blendRadius=0)
                    Set DigitalOutput pin=config_out[1]; digitalValue=0
                    barreno_actual := barreno_actual+1
                    SuppressedNode
                      Call Quitar_broca
                    SuppressedNode
                      Call Poner_broca
          Popup Message (haltProgram=false message=Linea14 con chica Terminada! inputType=Text)
          Folder Linea15
            Folder Marcar_puntos
              MoveL speed 100 mm/s, acceleration 500 mm/s^2 (useActiveTCP=true) feature=Base
                Waypoint Linea15_A: TCP in base x=626.307 y=508.675 z=110.445 mm, rx=-2.6326 ry=-1.7111 rz=-0.011 rad; joints [-145.159, -68.884, 100.875, -31.585, -220.372, 0.835] deg
                Waypoint Linea15_B: TCP in base x=626.328 y=587.416 z=110.05 mm, rx=-2.6327 ry=-1.711 rz=-0.011 rad; joints [-140.277, -63.781, 93.264, -29.039, -215.483, 0.889] deg
            Folder AB
              'desbaste_inicial'
              bajada_broca := p[0,0,-0.008,0,0,0]
              barrenos_menos1 := 3
              barreno_actual := 0
              Loop While (checkContinuously=false) expression=barreno_actual≤barrenos_menos1
                Folder Perforacion
                  MoveL speed 100 mm/s, acceleration 500 mm/s^2 (useActiveTCP=true) feature=Base
                    SuppressedNode
                      If barreno_actual≟3
                        barreno_actual := barreno_actual+1
                    internos := interpolate_pose(Linea15_A, Linea15_B, barreno_actual/barrenos_menos1)
                    Waypoint Waypoint (Variable): variable=internos
                    'desbaste_inicial'
                    bajada_broca := p[0,0,-0.008,0,0,0]
                    bajada := p[0,0,0.008,0,0,0]
                    MoveDirectionNode (selectedDirection=ZMinus toolParams=0.1, 0.15)
                      Until DISTANCE (allowActions=false deceleration=3 distanceNodeType=STOP) Distance=0.071; motionParameters(blendRadius=0)
                    MoveDirectionNode (selectedDirection=ZMinus toolParams=0.001, 0.001)
                      Until TOOL_CONTACT_DETECTION (allowActions=false retraction=0 decelerationAcceleration=0.001 decelerationAngularAcceleration=34.906585)
                    Popup Message (haltProgram=false message=punto contacto alanzdo inputType=Text)
                    MoveDirectionNode (selectedDirection=ZPlus toolParams=0.003, 0.005)
                      Until DISTANCE (allowActions=false deceleration=3 distanceNodeType=STOP) Distance=0.002; motionParameters(blendRadius=0)
                    Wait Sleep waitTime=0.3
                    Set DigitalOutput pin=config_out[1]; digitalValue=1
                    Wait Sleep waitTime=0.3
                    SuppressedNode
                      Loop Counting (count=3) loopVariable(name=Loop_86)
                        bajar := pose_add(get_actual_tcp_pose(), bajada_broca)
                        Waypoint Waypoint (Variable): motionParameters(jointSpeed=1.047198 jointAcceleration=1.396263 cartesianSpeed=0.001 cartesianAcceleration=0.005); variable=bajar
                        subir := pose_sub(get_actual_tcp_pose(), bajada_broca)
                        Waypoint Waypoint (Variable): motionParameters(jointSpeed=1.047198 jointAcceleration=1.396263 cartesianSpeed=0.005 cartesianAcceleration=0.01); variable=subir
                        bajada_broca := pose_sub(bajada_broca, bajada)
                    MoveDirectionNode (selectedDirection=ZPlus toolParams=0.1, 0.15)
                      Until DISTANCE (allowActions=false deceleration=3 distanceNodeType=STOP) Distance=0.08; motionParameters(blendRadius=0)
                    Set DigitalOutput pin=config_out[1]; digitalValue=0
                    barreno_actual := barreno_actual+1
                    SuppressedNode
                      Call Quitar_broca
                    SuppressedNode
                      Call Poner_broca
          Popup Message (haltProgram=false message=Linea15 con chica Terminada! inputType=Text)
          Folder Linea16
            Folder Marcar_puntos
              MoveL speed 100 mm/s, acceleration 500 mm/s^2 (useActiveTCP=true) feature=Base
                Waypoint Linea16_A: TCP in base x=464.714 y=611.413 z=110.697 mm, rx=-1.5443 ry=-2.7321 rz=-0.0069 rad; joints [-140.663, -77.848, 113.101, -34.922, -270.882, 0.394] deg; TCP offset x=0.411 y=-218.298 z=37.994 mm, rx=1.558 ry=-0.1255 rz=0.1212 rad
                Waypoint Linea16_B: TCP in base x=487.741 y=611.018 z=110.415 mm, rx=-1.5443 ry=-2.7321 rz=-0.0069 rad; joints [-142.061, -76.715, 111.675, -34.628, -272.279, 0.386] deg
            Folder AB
              'desbaste_inicial'
              bajada_broca := p[0,0,-0.008,0,0,0]
              barrenos_menos1 := 1
              barreno_actual := 0
              Loop While (checkContinuously=false) expression=barreno_actual≤barrenos_menos1
                Folder Perforacion
                  MoveL speed 100 mm/s, acceleration 500 mm/s^2 (useActiveTCP=true) feature=Base
                    SuppressedNode
                      If barreno_actual≟3
                        barreno_actual := barreno_actual+1
                    internos := interpolate_pose(Linea16_A, Linea16_B, barreno_actual/barrenos_menos1)
                    Waypoint Waypoint (Variable): variable=internos
                    'desbaste_inicial'
                    bajada_broca := p[0,0,-0.008,0,0,0]
                    bajada := p[0,0,0.008,0,0,0]
                    MoveDirectionNode (selectedDirection=ZMinus toolParams=0.1, 0.15)
                      Until DISTANCE (allowActions=false deceleration=3 distanceNodeType=STOP) Distance=0.071; motionParameters(blendRadius=0)
                    MoveDirectionNode (selectedDirection=ZMinus toolParams=0.001, 0.001)
                      Until TOOL_CONTACT_DETECTION (allowActions=false retraction=0 decelerationAcceleration=0.001 decelerationAngularAcceleration=34.906585)
                    Popup Message (haltProgram=false message=punto contacto alanzdo inputType=Text)
                    MoveDirectionNode (selectedDirection=ZPlus toolParams=0.003, 0.005)
                      Until DISTANCE (allowActions=false deceleration=3 distanceNodeType=STOP) Distance=0.002; motionParameters(blendRadius=0)
                    Wait Sleep waitTime=0.3
                    Set DigitalOutput pin=config_out[1]; digitalValue=1
                    Wait Sleep waitTime=0.3
                    SuppressedNode
                      Loop Counting (count=3) loopVariable(name=Loop_88)
                        bajar := pose_add(get_actual_tcp_pose(), bajada_broca)
                        Waypoint Waypoint (Variable): motionParameters(jointSpeed=1.047198 jointAcceleration=1.396263 cartesianSpeed=0.001 cartesianAcceleration=0.005); variable=bajar
                        subir := pose_sub(get_actual_tcp_pose(), bajada_broca)
                        Waypoint Waypoint (Variable): motionParameters(jointSpeed=1.047198 jointAcceleration=1.396263 cartesianSpeed=0.005 cartesianAcceleration=0.01); variable=subir
                        bajada_broca := pose_sub(bajada_broca, bajada)
                    MoveDirectionNode (selectedDirection=ZPlus toolParams=0.1, 0.15)
                      Until DISTANCE (allowActions=false deceleration=3 distanceNodeType=STOP) Distance=0.08; motionParameters(blendRadius=0)
                    Set DigitalOutput pin=config_out[1]; digitalValue=0
                    barreno_actual := barreno_actual+1
                    SuppressedNode
                      Call Quitar_broca
                    SuppressedNode
                      Call Poner_broca
          Popup Message (haltProgram=false message=Linea16 con chica Terminada! inputType=Text)
          Folder Linea17
            Folder Marcar_puntos
              MoveL speed 100 mm/s, acceleration 500 mm/s^2 (useActiveTCP=true) feature=Base
                Waypoint Linea17_A: TCP in base x=517.384 y=611.103 z=110.729 mm, rx=-1.5448 ry=-2.7327 rz=-0.0099 rad; joints [-143.713, -75.238, 109.731, -34.279, -273.925, 0.383] deg
                Waypoint Linea17_B: TCP in base x=569.253 y=610.697 z=110.46 mm, rx=-1.5448 ry=-2.7327 rz=-0.0099 rad; joints [-146.385, -72.438, 105.956, -33.3, -276.596, 0.373] deg
            Folder AB
              'desbaste_inicial'
              bajada_broca := p[0,0,-0.008,0,0,0]
              barrenos_menos1 := 2
              barreno_actual := 0
              Loop While (checkContinuously=false) expression=barreno_actual≤barrenos_menos1
                Folder Perforacion
                  MoveL speed 100 mm/s, acceleration 500 mm/s^2 (useActiveTCP=true) feature=Base
                    SuppressedNode
                      If barreno_actual≟3
                        barreno_actual := barreno_actual+1
                    internos := interpolate_pose(Linea17_A, Linea17_B, barreno_actual/barrenos_menos1)
                    Waypoint Waypoint (Variable): variable=internos
                    'desbaste_inicial'
                    bajada_broca := p[0,0,-0.008,0,0,0]
                    bajada := p[0,0,0.008,0,0,0]
                    MoveDirectionNode (selectedDirection=ZMinus toolParams=0.1, 0.15)
                      Until DISTANCE (allowActions=false deceleration=3 distanceNodeType=STOP) Distance=0.071; motionParameters(blendRadius=0)
                    MoveDirectionNode (selectedDirection=ZMinus toolParams=0.001, 0.001)
                      Until TOOL_CONTACT_DETECTION (allowActions=false retraction=0 decelerationAcceleration=0.001 decelerationAngularAcceleration=34.906585)
                    Popup Message (haltProgram=false message=punto contacto alanzdo inputType=Text)
                    MoveDirectionNode (selectedDirection=ZPlus toolParams=0.1, 0.15)
                      Until DISTANCE (allowActions=false deceleration=3 distanceNodeType=STOP) Distance=0.002; motionParameters(blendRadius=0)
                    Wait Sleep waitTime=0.3
                    Set DigitalOutput pin=config_out[1]; digitalValue=1
                    Wait Sleep waitTime=0.3
                    SuppressedNode
                      Loop Counting (count=3) loopVariable=Loop_90
                        bajar := pose_add(get_actual_tcp_pose(), bajada_broca)
                        Waypoint Waypoint (Variable): motionParameters(jointSpeed=1.047198 jointAcceleration=1.396263 cartesianSpeed=0.001 cartesianAcceleration=0.005); variable=bajar
                        subir := pose_sub(get_actual_tcp_pose(), bajada_broca)
                        Waypoint Waypoint (Variable): motionParameters(jointSpeed=1.047198 jointAcceleration=1.396263 cartesianSpeed=0.005 cartesianAcceleration=0.01); variable=subir
                        bajada_broca := pose_sub(bajada_broca, bajada)
                    MoveDirectionNode (selectedDirection=ZPlus toolParams=0.03, 0.035)
                      Until DISTANCE (allowActions=false deceleration=3 distanceNodeType=STOP) Distance=0.08; motionParameters(blendRadius=0)
                    Set DigitalOutput pin=config_out[1]; digitalValue=0
                    barreno_actual := barreno_actual+1
                    SuppressedNode
                      Call Quitar_broca
                    SuppressedNode
                      Call Poner_broca
          Popup Message (haltProgram=false message=Linea17 con chica Terminada! inputType=Text)
          Folder Linea18
            Folder Marcar_puntos
              MoveL speed 100 mm/s, acceleration 500 mm/s^2 (useActiveTCP=true) feature=Base
                Waypoint Linea18_A: TCP in base x=652.275 y=616.966 z=110.402 mm, rx=-1.5443 ry=-2.7321 rz=-0.0069 rad; joints [-149.578, -67.211, 98.412, -30.856, -279.791, 0.343] deg
